(*R8 ------------------------*)
		(*Input Data*)
		R8.FB_In.Robot_Type:=KUKA_KRC4_SAFEOP;
		R8.FB_In.Install_Zero_Orientation:= 0; 	(*Set this value between 0 and 359 to set the zero position of the robot physical install with reference to 12 o'clock symbol on UI screens*)
		R8.FB_In.Under_Construction:= GTAC_CONFIG.Under_Construction;
		R8.FB_In.In_SIM_Mode:= GTAC_CONFIG.In_SIM_Mode;
		R8.FB_In.SIM_StartWorkAround:= FALSE;  (*Main.SIM_WorkAround_StartRobots*)
		R8.FB_In.CoE_Read_Trigger:= (GTAC_CONFIG.Option_Robot_Count>=8) AND Pulse_CoERead;
		R8.FB_In.Ecat_Master_AmsNetID:= MAIN.ECAT_Master.AmsID;
		R8.FB_In.Prev_EcatNode_Present:= NOT R7.EK1100_NotPresent; (*Ensure Previous Node Exists to determine Ecat Cable Break of this Devices Input Cable*)
		R8.FB_In.Safety_RST:=SAFETY_RESET;
		R8.FB_In.Enable_Motion:= All_Estops_OK OR GTAC_CONFIG.Under_Construction;
		R8.FB_In.Alarm_RST:=In_From_ICxx.ControlPower1;
		R8.FB_In.Select_Play:=FALSE;
		R8.FB_In.Select_Teach:=FALSE;
		R8.FB_In.Select_Remote:=FALSE;
		R8.FB_In.Start_Scan:=In_From_ICxx.StartRobots;
		R8.FB_In.Stop_Scan:=In_From_ICxx.StopRobots;
		R8.FB_In.Stop_Scan2:=FALSE;
		R8.FB_In.In_DryCycle:= GTAC_CONFIG.Dry_Cycle_Enabled;
		R8.FB_In.Low_Speed:= GTAC_CONFIG.Low_Speed_Enabled;
		R8.FB_In.Speed_Request:= In_From_ICxx.Global_Robot_Speed;
		R8.FB_In.Force_MasterTest_Req:= Cell_Services_Prog.Human_Reqs_MasterTest OR Cell_Services_Prog.A_Robot_Reqs_MasterTest;
		R8.FB_In.Force_BrakeTest_Req:= Cell_Services_Prog.Human_Reqs_BrakeTest OR Cell_Services_Prog.A_Robot_Reqs_BrakeTest;
		R8.FB_In.Major_Faults:= Faults.System_Major_Fault;
		R8.FB_In.Teach_Interlock:=R8_Data.Teach_Interlock;
		R8.FB_In.Weld_Inhibit:=In_From_ICxx.Rxx_Weld_Inhibit;
		R8.FB_In.Option_Disable_WaterFLT:= FALSE AND GTAC_CONFIG.Under_Construction OR (MAIN.R8.Task_ID_Ack=Tip_Change_EXT); (*Used to disable water fault if no water is present. use with caution*)
		R8.FB_In.OK_ToEnter_EquipInterf1:=R8_Data.OK_ToEnter_EquipInterf1;
		R8.FB_In.OK_ToEnter_EquipInterf2:=R8_Data.OK_ToEnter_EquipInterf2;
		R8.FB_In.OK_ToEnter_EquipInterf3:=R8_Data.OK_ToEnter_EquipInterf3;
		R8.FB_In.OK_ToEnter_EquipInterf4:=R8_Data.OK_ToEnter_EquipInterf4;
		R8.FB_In.OK_ToEnter_EquipInterf5:=R8_Data.OK_ToEnter_EquipInterf5;
		R8.FB_In.OK_ToEnter_EquipInterf6:=R8_Data.OK_ToEnter_EquipInterf6;
		R8.FB_In.OK_ToEnter_EquipInterf7:=R8_Data.OK_ToEnter_EquipInterf7;
		R8.FB_In.OK_ToEnter_EquipInterf8:=R8_Data.OK_ToEnter_EquipInterf8;
		R8.FB_In.OK_ToEnter_EquipInterf9:=R8_Data.OK_ToEnter_EquipInterf9;
		R8.FB_In.OK_ToEnter_HumanInterf1:=R8_Data.OK_ToEnter_HumanInterf1;
		R8.FB_In.OK_ToEnter_HumanInterf2:=R8_Data.OK_ToEnter_HumanInterf2;
		R8.FB_In.OK_ToEnter_HumanInterf3:=R8_Data.OK_ToEnter_HumanInterf3;
		R8.FB_In.OK_ToEnter_HumanInterf4:=R8_Data.OK_ToEnter_HumanInterf4;
		R8.FB_In.OK_ToEnter_HumanInterf5:=R8_Data.OK_ToEnter_HumanInterf5;
		R8.FB_In.OK_ToEnter_HumanInterf6:=R8_Data.OK_ToEnter_HumanInterf6;
		R8.FB_In.OK_ToEnter_HumanInterf7:=R8_Data.OK_ToEnter_HumanInterf7;
		R8.FB_In.OK_ToEnter_HumanInterf8:=R8_Data.OK_ToEnter_HumanInterf8;
		R8.FB_In.OK_ToEnter_RobotInterfs:= R8_Data.OK_ToEnter_RobotInterfs;
		R8.FB_In.Fix_ID:=R8_Data.Fix_ID[R8.Location_Index];
		R8.FB_In.Model_ID:=R8_Data.Model_ID[R8.Location_Index];
		R8.FB_In.Task_ID:=R8_Data.Task_ID[R8.Location_Index];
		R8.FB_In.Proceed_From_Pounce:=R8_Data.Proceed_From_Pounce[R8.Location_Index];
		R8.FB_In.Complete_Ack:=R8_Data.Complete_Ack[R8.Location_Index];
		R8.FB_In.PeripheralReq_Ack:=R8_Data.PeripheralReq_Ack[R8.Location_Index];
		R8.FB_In.AuxReq_Ack:=R8_Data.AuxReq_Ack[R8.Location_Index];
		R8.FB_In.User_Inputs.0:= FALSE;
		R8.FB_In.User_Inputs.1:= FALSE;
		R8.FB_In.User_Inputs.2:= FALSE;
		R8.FB_In.User_Inputs.3:= FALSE;
		R8.FB_In.User_Inputs.4:= FALSE;
		R8.FB_In.User_Inputs.5:= FALSE;
		R8.FB_In.User_Inputs.6:= FALSE;
		R8.FB_In.User_Inputs.7:= FALSE;
			(*Configure Options Amounts*)
			R8.FB_In.Options.WeldCont_Amount:= 0; 					(*Select amount of Spot Type Weld Controllers here (0 min, 4 max)*)
			R8.FB_In.Options.WaterStand_Amount:= 0;				(*Select amount of Water Stands here (0 min, 2 max)*)
			R8.FB_In.Options.MIGCont_Amount:= 1;					(*Select amount of MIG Type Weld Controllers here (0 min, 1 max)*)
			R8.FB_In.Options.Reamer_Amount:= 1;					(*Select amount of Tip Reamers here (0 min, 1 max)*)
			R8.FB_In.Options.EOAT_Amount:= 0;						(*Assign EOAT number to robot (0 min, 10 max)*)
			(*Configure Options Parameters*)
			
			R8.Reamer[1](
				(*FB Inputs*)
					Enable_Motion:= All_Estops_OK,
					Fronius_Ream:= TRUE,
                    Binzel_Ream:= FALSE,  (*optional*)
					
					Ream_REQ:= R8.Peripheral_Req.1 AND ((R8.Task_ID_Ack=Tip_Dress)OR (R8.In_T1 AND R8.Peripheral_Req.5)),
					Ream_Time:= T#2S,
					Ream_Clamp_Open:= R8.Reamer[1].N01.I.1,
					Spray_REQ:= R8.Peripheral_Req.2 AND ((R8.Task_ID_Ack=Tip_Dress)OR (R8.In_T1 AND R8.Peripheral_Req.5)),
					Spray_Time:= T#2S,
					F_WireCutter_REQ:= R8.Peripheral_Req.4 AND ((R8.Task_ID_Ack=Tip_Dress)OR (R8.In_T1 AND R8.Peripheral_Req.5)),
					F_WireCutter_Time:= T#1S,
					
				(*FB Outputs*)
					Reaming_Complete=> ,(*mapped in cell services*)
					(*The following are for Binzel type reamers only*)
					LifterUp_ACK=> , (*mapped in cell services*)
					Clamp_ACK=>,(*mapped in cell services*)
					Injector_ACK=> ,(*mapped in cell services*)
					WireCutter_ACK=> (*mapped in cell services*)
					);
			(*R8.Reamer[1](
				(*FB Inputs*)
					Enable_Motion:= All_Estops_OK,
					Fronius_Ream:= TRUE,
                    Binzel_Ream:= FALSE,  (*optional*)
					Ream_REQ:= R8.Peripheral_Req.5 AND (R8.Task_ID_Ack=Tip_Dress),

				(*FB Outputs*)
					Reaming_Complete=> ,(*mapped in cell services*)
					);*)
		(*Call Actual Object*)
		R8();
		(*Output Data*)
		Out_To_ICxx.Robot[8].Robot_Type:= R8.FB_In.Robot_Type;
		Out_To_ICxx.Robot[8].Status:= R8.Status;
		Out_To_ICxx.Robot[8].Axis_Data[1]:= R8.S_Axis_Pos_Raw;
		Out_To_ICxx.Robot[8].In_Image:= R8.Input_Image;
		Out_To_ICxx.Robot[8].Out_Image:= R8.Output_Image;
		Out_To_ICxx.Robot[8].Discrete_ImageFSOE:= R8.Discrete_Image_FSoE;
		Out_To_ICxx.Robot[8].Options:= R8.FB_In.Options;
			Out_To_ICxx.Robot[8].WS_Discrete_Image[1]:= R8.WS[1].Discrete_Image;
			Out_To_ICxx.Robot[8].WS_Discrete_Image[2]:= R8.WS[2].Discrete_Image;
 			Out_To_ICxx.Robot[8].ATI_Discrete_Image:= R8.ATI[1].Discrete_Image;
			Out_To_ICxx.Robot[8].Reamer_Discrete_Image:= R8.Reamer[1].Discrete_Image;
			Out_To_ICxx.Robot[8].Fronius_Status:= R8.Fronius_Status;
		Out_To_ICxx.Robot[8].Ped_IO_ToShow[1]:= 0;			(*Set to Ped value if this robots ecat string contains the Ped's IO*)
		Out_To_ICxx.Robot[8].Ped_IO_ToShow[2]:= 0;			(*Set to Ped value if this robots ecat string contains the Ped's IO*)
		Out_To_ICxx.Robot[8].ECAT_Cable_Breaks:= R8.ECatSlave_Cable_Breaks;
		Out_To_ICxx.Robot[8].CT:= R8.CT;



(*R9 ------------------------*)
		(*Input Data*)
		R9.FB_In.Robot_Type:=KUKA_KRC4_SAFEOP;
		R9.FB_In.Install_Zero_Orientation:= 0; 	(*Set this value between 0 and 359 to set the zero position of the robot physical install with reference to 12 o'clock symbol on UI screens*)
		R9.FB_In.Under_Construction:= GTAC_CONFIG.Under_Construction;
		R9.FB_In.In_SIM_Mode:= GTAC_CONFIG.In_SIM_Mode;
		R9.FB_In.SIM_StartWorkAround:= FALSE;  (*Main.SIM_WorkAround_StartRobots*)
		R9.FB_In.CoE_Read_Trigger:= (GTAC_CONFIG.Option_Robot_Count>=9) AND Pulse_CoERead;
		R9.FB_In.Ecat_Master_AmsNetID:= MAIN.ECAT_Master.AmsID;
		R9.FB_In.Prev_EcatNode_Present:= NOT R8.EK1100_NotPresent; (*Ensure Previous Node Exists to determine Ecat Cable Break of this Devices Input Cable*)
		R9.FB_In.Safety_RST:=SAFETY_RESET;
		R9.FB_In.Enable_Motion:= All_Estops_OK OR GTAC_CONFIG.Under_Construction;
		R9.FB_In.Alarm_RST:=In_From_ICxx.ControlPower1;
		R9.FB_In.Select_Play:=FALSE;
		R9.FB_In.Select_Teach:=FALSE;
		R9.FB_In.Select_Remote:=FALSE;
		R9.FB_In.Start_Scan:=In_From_ICxx.StartRobots;
		R9.FB_In.Stop_Scan:=In_From_ICxx.StopRobots;
		R9.FB_In.Stop_Scan2:=FALSE;
		R9.FB_In.In_DryCycle:= GTAC_CONFIG.Dry_Cycle_Enabled;
		R9.FB_In.Low_Speed:= GTAC_CONFIG.Low_Speed_Enabled;
		R9.FB_In.Speed_Request:= In_From_ICxx.Global_Robot_Speed;
		R9.FB_In.Force_MasterTest_Req:= Cell_Services_Prog.Human_Reqs_MasterTest OR Cell_Services_Prog.A_Robot_Reqs_MasterTest;
		R9.FB_In.Force_BrakeTest_Req:= Cell_Services_Prog.Human_Reqs_BrakeTest OR Cell_Services_Prog.A_Robot_Reqs_BrakeTest;
		R9.FB_In.Major_Faults:= Faults.System_Major_Fault;
		R9.FB_In.Teach_Interlock:=R9_Data.Teach_Interlock;
		R9.FB_In.Weld_Inhibit:=In_From_ICxx.Rxx_Weld_Inhibit;
		R9.FB_In.Option_Disable_WaterFLT:= FALSE AND GTAC_CONFIG.Under_Construction OR (MAIN.R9.Task_ID_Ack=Tip_Change_EXT); (*Used to disable water fault if no water is present. use with caution*)
		R9.FB_In.OK_ToEnter_EquipInterf1:=R9_Data.OK_ToEnter_EquipInterf1;
		R9.FB_In.OK_ToEnter_EquipInterf2:=R9_Data.OK_ToEnter_EquipInterf2;
		R9.FB_In.OK_ToEnter_EquipInterf3:=R9_Data.OK_ToEnter_EquipInterf3;
		R9.FB_In.OK_ToEnter_EquipInterf4:=R9_Data.OK_ToEnter_EquipInterf4;
		R9.FB_In.OK_ToEnter_EquipInterf5:=R9_Data.OK_ToEnter_EquipInterf5;
		R9.FB_In.OK_ToEnter_EquipInterf6:=R9_Data.OK_ToEnter_EquipInterf6;
		R9.FB_In.OK_ToEnter_EquipInterf7:=R9_Data.OK_ToEnter_EquipInterf7;
		R9.FB_In.OK_ToEnter_EquipInterf8:=R9_Data.OK_ToEnter_EquipInterf8;
		R9.FB_In.OK_ToEnter_EquipInterf9:=R9_Data.OK_ToEnter_EquipInterf9;
		R9.FB_In.OK_ToEnter_HumanInterf1:=R9_Data.OK_ToEnter_HumanInterf1;
		R9.FB_In.OK_ToEnter_HumanInterf2:=R9_Data.OK_ToEnter_HumanInterf2;
		R9.FB_In.OK_ToEnter_HumanInterf3:=R9_Data.OK_ToEnter_HumanInterf3;
		R9.FB_In.OK_ToEnter_HumanInterf4:=R9_Data.OK_ToEnter_HumanInterf4;
		R9.FB_In.OK_ToEnter_HumanInterf5:=R9_Data.OK_ToEnter_HumanInterf5;
		R9.FB_In.OK_ToEnter_HumanInterf6:=R9_Data.OK_ToEnter_HumanInterf6;
		R9.FB_In.OK_ToEnter_HumanInterf7:=R9_Data.OK_ToEnter_HumanInterf7;
		R9.FB_In.OK_ToEnter_HumanInterf8:=R9_Data.OK_ToEnter_HumanInterf8;
		R9.FB_In.OK_ToEnter_RobotInterfs:= R9_Data.OK_ToEnter_RobotInterfs;
		R9.FB_In.Fix_ID:=R9_Data.Fix_ID[R9.Location_Index];
		R9.FB_In.Model_ID:=R9_Data.Model_ID[R9.Location_Index];
		R9.FB_In.Task_ID:=R9_Data.Task_ID[R9.Location_Index];
		R9.FB_In.Proceed_From_Pounce:=R9_Data.Proceed_From_Pounce[R9.Location_Index];
		R9.FB_In.Complete_Ack:=R9_Data.Complete_Ack[R9.Location_Index];
		R9.FB_In.PeripheralReq_Ack:=R9_Data.PeripheralReq_Ack[R9.Location_Index];
		R9.FB_In.AuxReq_Ack:=R9_Data.AuxReq_Ack[R9.Location_Index];
		R9.FB_In.User_Inputs.0:= FALSE;
		R9.FB_In.User_Inputs.1:= FALSE;
		R9.FB_In.User_Inputs.2:= FALSE;
		R9.FB_In.User_Inputs.3:= FALSE;
		R9.FB_In.User_Inputs.4:= FALSE;
		R9.FB_In.User_Inputs.5:= FALSE;
		R9.FB_In.User_Inputs.6:= FALSE;
		R9.FB_In.User_Inputs.7:= FALSE;
			(*Configure Options Amounts*)
			R9.FB_In.Options.WeldCont_Amount:= 0; 					(*Select amount of Spot Type Weld Controllers here (0 min, 4 max)*)
			R9.FB_In.Options.WaterStand_Amount:= 0;				(*Select amount of Water Stands here (0 min, 2 max)*)
			R9.FB_In.Options.MIGCont_Amount:= 1;					(*Select amount of MIG Type Weld Controllers here (0 min, 1 max)*)
			R9.FB_In.Options.Reamer_Amount:= 1;					(*Select amount of Tip Reamers here (0 min, 1 max)*)
			R9.FB_In.Options.EOAT_Amount:= 0;						(*Assign EOAT number to robot (0 min, 10 max)*)
			(*Configure Options Parameters*)
			
			R9.Reamer[1](
				(*FB Inputs*)
					Enable_Motion:= All_Estops_OK,
					Fronius_Ream:= TRUE,
                    Binzel_Ream:= FALSE,  (*optional*)
					
					Ream_REQ:= R9.Peripheral_Req.1 AND ((R9.Task_ID_Ack=Tip_Dress)OR (R9.In_T1 AND R9.Peripheral_Req.5)),
					Ream_Time:= T#2S,
					Ream_Clamp_Open:= R9.Reamer[1].N01.I.1,
					Spray_REQ:= R9.Peripheral_Req.2 AND ((R9.Task_ID_Ack=Tip_Dress)OR (R9.In_T1 AND R9.Peripheral_Req.5)),
					Spray_Time:= T#2S,
					F_WireCutter_REQ:= R9.Peripheral_Req.4 AND ((R9.Task_ID_Ack=Tip_Dress)OR (R9.In_T1 AND R9.Peripheral_Req.5)),
					F_WireCutter_Time:= T#1S,
					
				(*FB Outputs*)
					Reaming_Complete=> ,(*mapped in cell services*)
					(*The following are for Binzel type reamers only*)
					LifterUp_ACK=> , (*mapped in cell services*)
					Clamp_ACK=>,(*mapped in cell services*)
					Injector_ACK=> ,(*mapped in cell services*)
					WireCutter_ACK=> (*mapped in cell services*)
					);
			(*R9.Reamer[1](
				(*FB Inputs*)
					Enable_Motion:= All_Estops_OK,
					Fronius_Ream:= TRUE,
                    Binzel_Ream:= FALSE,  (*optional*)
					Ream_REQ:= R9.Peripheral_Req.5 AND (R9.Task_ID_Ack=Tip_Dress),

				(*FB Outputs*)
					Reaming_Complete=> ,(*mapped in cell services*)
					);*)
		(*Call Actual Object*)
		R9();
		(*Output Data*)
		Out_To_ICxx.Robot[9].Robot_Type:= R9.FB_In.Robot_Type;
		Out_To_ICxx.Robot[9].Status:= R9.Status;
		Out_To_ICxx.Robot[9].Axis_Data[1]:= R9.S_Axis_Pos_Raw;
		Out_To_ICxx.Robot[9].In_Image:= R9.Input_Image;
		Out_To_ICxx.Robot[9].Out_Image:= R9.Output_Image;
		Out_To_ICxx.Robot[9].Discrete_ImageFSOE:= R9.Discrete_Image_FSoE;
		Out_To_ICxx.Robot[9].Options:= R9.FB_In.Options;
			Out_To_ICxx.Robot[9].WS_Discrete_Image[1]:= R9.WS[1].Discrete_Image;
			Out_To_ICxx.Robot[9].WS_Discrete_Image[2]:= R9.WS[2].Discrete_Image;
 			Out_To_ICxx.Robot[9].ATI_Discrete_Image:= R9.ATI[1].Discrete_Image;
			Out_To_ICxx.Robot[9].Reamer_Discrete_Image:= R9.Reamer[1].Discrete_Image;
			Out_To_ICxx.Robot[9].Fronius_Status:= R9.Fronius_Status;
		Out_To_ICxx.Robot[9].Ped_IO_ToShow[1]:= 0;			(*Set to Ped value if this robots ecat string contains the Ped's IO*)
		Out_To_ICxx.Robot[9].Ped_IO_ToShow[2]:= 0;			(*Set to Ped value if this robots ecat string contains the Ped's IO*)
		Out_To_ICxx.Robot[9].ECAT_Cable_Breaks:= R9.ECatSlave_Cable_Breaks;
		Out_To_ICxx.Robot[9].CT:= R9.CT;



(*R10 ------------------------*)
		(*Input Data*)
		R10.FB_In.Robot_Type:=KUKA_KRC4_SAFEOP;
		R10.FB_In.Install_Zero_Orientation:= 0; 	(*Set this value between 0 and 359 to set the zero position of the robot physical install with reference to 12 o'clock symbol on UI screens*)
		R10.FB_In.Under_Construction:= GTAC_CONFIG.Under_Construction;
		R10.FB_In.In_SIM_Mode:= GTAC_CONFIG.In_SIM_Mode;
		R10.FB_In.SIM_StartWorkAround:= FALSE;  (*Main.SIM_WorkAround_StartRobots*)
		R10.FB_In.CoE_Read_Trigger:= (GTAC_CONFIG.Option_Robot_Count>=10) AND Pulse_CoERead;
		R10.FB_In.Ecat_Master_AmsNetID:= MAIN.ECAT_Master.AmsID;
		R10.FB_In.Prev_EcatNode_Present:= NOT R9.EK1100_NotPresent; (*Ensure Previous Node Exists to determine Ecat Cable Break of this Devices Input Cable*)
		R10.FB_In.Safety_RST:=SAFETY_RESET;
		R10.FB_In.Enable_Motion:= All_Estops_OK OR GTAC_CONFIG.Under_Construction;
		R10.FB_In.Alarm_RST:=In_From_ICxx.ControlPower1;
		R10.FB_In.Select_Play:=FALSE;
		R10.FB_In.Select_Teach:=FALSE;
		R10.FB_In.Select_Remote:=FALSE;
		R10.FB_In.Start_Scan:=In_From_ICxx.StartRobots;
		R10.FB_In.Stop_Scan:=In_From_ICxx.StopRobots;
		R10.FB_In.Stop_Scan2:=FALSE;
		R10.FB_In.In_DryCycle:= GTAC_CONFIG.Dry_Cycle_Enabled;
		R10.FB_In.Low_Speed:= GTAC_CONFIG.Low_Speed_Enabled;
		R10.FB_In.Speed_Request:= In_From_ICxx.Global_Robot_Speed;
		R10.FB_In.Force_MasterTest_Req:= Cell_Services_Prog.Human_Reqs_MasterTest OR Cell_Services_Prog.A_Robot_Reqs_MasterTest;
		R10.FB_In.Force_BrakeTest_Req:= Cell_Services_Prog.Human_Reqs_BrakeTest OR Cell_Services_Prog.A_Robot_Reqs_BrakeTest;
		R10.FB_In.Major_Faults:= Faults.System_Major_Fault;
		R10.FB_In.Teach_Interlock:=R10_Data.Teach_Interlock;
		R10.FB_In.Weld_Inhibit:=In_From_ICxx.Rxx_Weld_Inhibit;
		R10.FB_In.Option_Disable_WaterFLT:= FALSE AND GTAC_CONFIG.Under_Construction OR (MAIN.R10.Task_ID_Ack=Tip_Change_EXT); (*Used to disable water fault if no water is present. use with caution*)
		R10.FB_In.OK_ToEnter_EquipInterf1:=R10_Data.OK_ToEnter_EquipInterf1;
		R10.FB_In.OK_ToEnter_EquipInterf2:=R10_Data.OK_ToEnter_EquipInterf2;
		R10.FB_In.OK_ToEnter_EquipInterf3:=R10_Data.OK_ToEnter_EquipInterf3;
		R10.FB_In.OK_ToEnter_EquipInterf4:=R10_Data.OK_ToEnter_EquipInterf4;
		R10.FB_In.OK_ToEnter_EquipInterf5:=R10_Data.OK_ToEnter_EquipInterf5;
		R10.FB_In.OK_ToEnter_EquipInterf6:=R10_Data.OK_ToEnter_EquipInterf6;
		R10.FB_In.OK_ToEnter_EquipInterf7:=R10_Data.OK_ToEnter_EquipInterf7;
		R10.FB_In.OK_ToEnter_EquipInterf8:=R10_Data.OK_ToEnter_EquipInterf8;
		R10.FB_In.OK_ToEnter_EquipInterf9:=R10_Data.OK_ToEnter_EquipInterf9;
		R10.FB_In.OK_ToEnter_HumanInterf1:=R10_Data.OK_ToEnter_HumanInterf1;
		R10.FB_In.OK_ToEnter_HumanInterf2:=R10_Data.OK_ToEnter_HumanInterf2;
		R10.FB_In.OK_ToEnter_HumanInterf3:=R10_Data.OK_ToEnter_HumanInterf3;
		R10.FB_In.OK_ToEnter_HumanInterf4:=R10_Data.OK_ToEnter_HumanInterf4;
		R10.FB_In.OK_ToEnter_HumanInterf5:=R10_Data.OK_ToEnter_HumanInterf5;
		R10.FB_In.OK_ToEnter_HumanInterf6:=R10_Data.OK_ToEnter_HumanInterf6;
		R10.FB_In.OK_ToEnter_HumanInterf7:=R10_Data.OK_ToEnter_HumanInterf7;
		R10.FB_In.OK_ToEnter_HumanInterf8:=R10_Data.OK_ToEnter_HumanInterf8;
		R10.FB_In.OK_ToEnter_RobotInterfs:= R10_Data.OK_ToEnter_RobotInterfs;
		R10.FB_In.Fix_ID:=R10_Data.Fix_ID[R10.Location_Index];
		R10.FB_In.Model_ID:=R10_Data.Model_ID[R10.Location_Index];
		R10.FB_In.Task_ID:=R10_Data.Task_ID[R10.Location_Index];
		R10.FB_In.Proceed_From_Pounce:=R10_Data.Proceed_From_Pounce[R10.Location_Index];
		R10.FB_In.Complete_Ack:=R10_Data.Complete_Ack[R10.Location_Index];
		R10.FB_In.PeripheralReq_Ack:=R10_Data.PeripheralReq_Ack[R10.Location_Index];
		R10.FB_In.AuxReq_Ack:=R10_Data.AuxReq_Ack[R10.Location_Index];
		R10.FB_In.User_Inputs.0:= FALSE;
		R10.FB_In.User_Inputs.1:= FALSE;
		R10.FB_In.User_Inputs.2:= FALSE;
		R10.FB_In.User_Inputs.3:= FALSE;
		R10.FB_In.User_Inputs.4:= FALSE;
		R10.FB_In.User_Inputs.5:= FALSE;
		R10.FB_In.User_Inputs.6:= FALSE;
		R10.FB_In.User_Inputs.7:= FALSE;
			(*Configure Options Amounts*)
			R10.FB_In.Options.WeldCont_Amount:= 0; 					(*Select amount of Spot Type Weld Controllers here (0 min, 4 max)*)
			R10.FB_In.Options.WaterStand_Amount:= 0;				(*Select amount of Water Stands here (0 min, 2 max)*)
			R10.FB_In.Options.MIGCont_Amount:= 1;					(*Select amount of MIG Type Weld Controllers here (0 min, 1 max)*)
			R10.FB_In.Options.Reamer_Amount:= 1;					(*Select amount of Tip Reamers here (0 min, 1 max)*)
			R10.FB_In.Options.EOAT_Amount:= 0;					(*Assign EOAT number to robot (0 min, 10 max)*)
			(*Configure Options Parameters*)
			(*R10.Reamer[1](
				(*FB Inputs*)
					Enable_Motion:= All_Estops_OK,
					Fronius_Ream:= TRUE,
                    Binzel_Ream:= FALSE,  (*optional*)
					Ream_REQ:= R10.Peripheral_Req.5 AND (R10.Task_ID_Ack=Tip_Dress),

				(*FB Outputs*)
					Reaming_Complete=> ,(*mapped in cell services*)
					);*)
		(*Call Actual Object*)
		R10();
		(*Output Data*)
		Out_To_ICxx.Robot[10].Robot_Type:= R10.FB_In.Robot_Type;
		(*To create less work, since there is no welding, changeing this number to 307 so we dont have to mess with the kuka FB, just screens. "us_Rxx_Status" - added 307 "inspecting"*)
		IF (R10.Status = 305) THEN
		Out_To_ICxx.Robot[10].Status:= 307; 
		ELSE
		Out_To_ICxx.Robot[10].Status:= R10.Status;
		END_IF
		Out_To_ICxx.Robot[10].Axis_Data[1]:= R10.S_Axis_Pos_Raw;
		Out_To_ICxx.Robot[10].In_Image:= R10.Input_Image;
		Out_To_ICxx.Robot[10].Out_Image:= R10.Output_Image;
		Out_To_ICxx.Robot[10].Discrete_ImageFSOE:= R10.Discrete_Image_FSoE;
		Out_To_ICxx.Robot[10].Options:= R10.FB_In.Options;
			Out_To_ICxx.Robot[10].WS_Discrete_Image[1]:= R10.WS[1].Discrete_Image;
			Out_To_ICxx.Robot[10].WS_Discrete_Image[2]:= R10.WS[2].Discrete_Image;
 			Out_To_ICxx.Robot[10].ATI_Discrete_Image:= R10.ATI[1].Discrete_Image;
			Out_To_ICxx.Robot[10].Reamer_Discrete_Image:= R10.Reamer[1].Discrete_Image;
			Out_To_ICxx.Robot[10].Fronius_Status:= R10.Fronius_Status;
		Out_To_ICxx.Robot[10].Ped_IO_ToShow[1]:= 0;			(*Set to Ped value if this robots ecat string contains the Ped's IO*)
		Out_To_ICxx.Robot[10].Ped_IO_ToShow[2]:= 0;			(*Set to Ped value if this robots ecat string contains the Ped's IO*)
		Out_To_ICxx.Robot[10].ECAT_Cable_Breaks:= R10.ECatSlave_Cable_Breaks;
		Out_To_ICxx.Robot[10].CT:= R10.CT;



(*R11 ------------------------*)
		(*Input Data*)
		R11.FB_In.Robot_Type:=KUKA_KRC4_SAFEOP;
		R11.FB_In.Install_Zero_Orientation:= 0; 	(*Set this value between 0 and 359 to set the zero position of the robot physical install with reference to 12 o'clock symbol on UI screens*)
		R11.FB_In.Under_Construction:= GTAC_CONFIG.Under_Construction;
		R11.FB_In.In_SIM_Mode:= GTAC_CONFIG.In_SIM_Mode;
		R11.FB_In.SIM_StartWorkAround:= FALSE;  (*Main.SIM_WorkAround_StartRobots*)
		R11.FB_In.CoE_Read_Trigger:= (GTAC_CONFIG.Option_Robot_Count>=11) AND Pulse_CoERead;
		R11.FB_In.Ecat_Master_AmsNetID:= MAIN.ECAT_Master.AmsID;
		R11.FB_In.Prev_EcatNode_Present:= NOT R10.EK1100_NotPresent; (*Ensure Previous Node Exists to determine Ecat Cable Break of this Devices Input Cable*)
		R11.FB_In.Safety_RST:=SAFETY_RESET;
		R11.FB_In.Enable_Motion:= All_Estops_OK OR GTAC_CONFIG.Under_Construction;
		R11.FB_In.Alarm_RST:=In_From_ICxx.ControlPower1;
		R11.FB_In.Select_Play:=FALSE;
		R11.FB_In.Select_Teach:=FALSE;
		R11.FB_In.Select_Remote:=FALSE;
		R11.FB_In.Start_Scan:=In_From_ICxx.StartRobots;
		R11.FB_In.Stop_Scan:=In_From_ICxx.StopRobots;
		R11.FB_In.Stop_Scan2:=FALSE;
		R11.FB_In.In_DryCycle:= GTAC_CONFIG.Dry_Cycle_Enabled;
		R11.FB_In.Low_Speed:= GTAC_CONFIG.Low_Speed_Enabled;
		R11.FB_In.Speed_Request:= In_From_ICxx.Global_Robot_Speed;
		R11.FB_In.Force_MasterTest_Req:= Cell_Services_Prog.Human_Reqs_MasterTest OR Cell_Services_Prog.A_Robot_Reqs_MasterTest;
		R11.FB_In.Force_BrakeTest_Req:= Cell_Services_Prog.Human_Reqs_BrakeTest OR Cell_Services_Prog.A_Robot_Reqs_BrakeTest;
		R11.FB_In.Major_Faults:= Faults.System_Major_Fault;
		R11.FB_In.Teach_Interlock:=R11_Data.Teach_Interlock;
		R11.FB_In.Weld_Inhibit:=In_From_ICxx.Rxx_Weld_Inhibit;
		R11.FB_In.Option_Disable_WaterFLT:= FALSE AND GTAC_CONFIG.Under_Construction OR (MAIN.R11.Task_ID_Ack=Tip_Change_EXT); (*Used to disable water fault if no water is present. use with caution*)
		R11.FB_In.OK_ToEnter_EquipInterf1:=R11_Data.OK_ToEnter_EquipInterf1;
		R11.FB_In.OK_ToEnter_EquipInterf2:=R11_Data.OK_ToEnter_EquipInterf2;
		R11.FB_In.OK_ToEnter_EquipInterf3:=R11_Data.OK_ToEnter_EquipInterf3;
		R11.FB_In.OK_ToEnter_EquipInterf4:=R11_Data.OK_ToEnter_EquipInterf4;
		R11.FB_In.OK_ToEnter_EquipInterf5:=R11_Data.OK_ToEnter_EquipInterf5;
		R11.FB_In.OK_ToEnter_EquipInterf6:=R11_Data.OK_ToEnter_EquipInterf6;
		R11.FB_In.OK_ToEnter_EquipInterf7:=R11_Data.OK_ToEnter_EquipInterf7;
		R11.FB_In.OK_ToEnter_EquipInterf8:=R11_Data.OK_ToEnter_EquipInterf8;
		R11.FB_In.OK_ToEnter_EquipInterf9:=R11_Data.OK_ToEnter_EquipInterf9;
		R11.FB_In.OK_ToEnter_HumanInterf1:=R11_Data.OK_ToEnter_HumanInterf1;
		R11.FB_In.OK_ToEnter_HumanInterf2:=R11_Data.OK_ToEnter_HumanInterf2;
		R11.FB_In.OK_ToEnter_HumanInterf3:=R11_Data.OK_ToEnter_HumanInterf3;
		R11.FB_In.OK_ToEnter_HumanInterf4:=R11_Data.OK_ToEnter_HumanInterf4;
		R11.FB_In.OK_ToEnter_HumanInterf5:=R11_Data.OK_ToEnter_HumanInterf5;
		R11.FB_In.OK_ToEnter_HumanInterf6:=R11_Data.OK_ToEnter_HumanInterf6;
		R11.FB_In.OK_ToEnter_HumanInterf7:=R11_Data.OK_ToEnter_HumanInterf7;
		R11.FB_In.OK_ToEnter_HumanInterf8:=R11_Data.OK_ToEnter_HumanInterf8;
		R11.FB_In.OK_ToEnter_RobotInterfs:= R11_Data.OK_ToEnter_RobotInterfs;
		R11.FB_In.Fix_ID:=R11_Data.Fix_ID[R11.Location_Index];
		R11.FB_In.Model_ID:=R11_Data.Model_ID[R11.Location_Index];
		R11.FB_In.Task_ID:=R11_Data.Task_ID[R11.Location_Index];
		R11.FB_In.Proceed_From_Pounce:=R11_Data.Proceed_From_Pounce[R11.Location_Index];
		R11.FB_In.Complete_Ack:=R11_Data.Complete_Ack[R11.Location_Index];
		R11.FB_In.PeripheralReq_Ack:=R11_Data.PeripheralReq_Ack[R11.Location_Index];
		R11.FB_In.AuxReq_Ack:=R11_Data.AuxReq_Ack[R11.Location_Index];
		R11.FB_In.User_Inputs.0:= FALSE;
		R11.FB_In.User_Inputs.1:= FALSE;
		R11.FB_In.User_Inputs.2:= FALSE;
		R11.FB_In.User_Inputs.3:= FALSE;
		R11.FB_In.User_Inputs.4:= FALSE;
		R11.FB_In.User_Inputs.5:= FALSE;
		R11.FB_In.User_Inputs.6:= FALSE;
		R11.FB_In.User_Inputs.7:= FALSE;
			(*Configure Options Amounts*)
			R11.FB_In.Options.WeldCont_Amount:= 0; 					(*Select amount of Spot Type Weld Controllers here (0 min, 4 max)*)
			R11.FB_In.Options.WaterStand_Amount:= 0;				(*Select amount of Water Stands here (0 min, 2 max)*)
			R11.FB_In.Options.MIGCont_Amount:= 1;					(*Select amount of MIG Type Weld Controllers here (0 min, 1 max)*)
			R11.FB_In.Options.Reamer_Amount:= 1;					(*Select amount of Tip Reamers here (0 min, 1 max)*)
			R11.FB_In.Options.EOAT_Amount:= 0;					(*Assign EOAT number to robot (0 min, 10 max)*)
			(*Configure Options Parameters*)
			(*R11.Reamer[1](
				(*FB Inputs*)
					Enable_Motion:= All_Estops_OK,
					Fronius_Ream:= TRUE,
                    Binzel_Ream:= FALSE,  (*optional*)
					Ream_REQ:= R11.Peripheral_Req.5 AND (R11.Task_ID_Ack=Tip_Dress),

				(*FB Outputs*)
					Reaming_Complete=> ,(*mapped in cell services*)
					);*)
		(*Call Actual Object*)
		R11();
		(*Output Data*)
		Out_To_ICxx.Robot[11].Robot_Type:= R11.FB_In.Robot_Type;
		(*To create less work, since there is no welding, changeing this number to 307 so we dont have to mess with the kuka FB, just screens. "us_Rxx_Status" - added 307 "inspecting"*)
		IF (R11.Status = 305) THEN
		Out_To_ICxx.Robot[11].Status:= 307; 
		ELSE
		Out_To_ICxx.Robot[11].Status:= R11.Status;
		END_IF
		Out_To_ICxx.Robot[11].Axis_Data[1]:= R11.S_Axis_Pos_Raw;
		Out_To_ICxx.Robot[11].In_Image:= R11.Input_Image;
		Out_To_ICxx.Robot[11].Out_Image:= R11.Output_Image;
		Out_To_ICxx.Robot[11].Discrete_ImageFSOE:= R11.Discrete_Image_FSoE;
		Out_To_ICxx.Robot[11].Options:= R11.FB_In.Options;
			Out_To_ICxx.Robot[11].WS_Discrete_Image[1]:= R11.WS[1].Discrete_Image;
			Out_To_ICxx.Robot[11].WS_Discrete_Image[2]:= R11.WS[2].Discrete_Image;
 			Out_To_ICxx.Robot[11].ATI_Discrete_Image:= R11.ATI[1].Discrete_Image;
			Out_To_ICxx.Robot[11].Reamer_Discrete_Image:= R11.Reamer[1].Discrete_Image;
			Out_To_ICxx.Robot[11].Fronius_Status:= R11.Fronius_Status;
		Out_To_ICxx.Robot[11].Ped_IO_ToShow[1]:= 0;			(*Set to Ped value if this robots ecat string contains the Ped's IO*)
		Out_To_ICxx.Robot[11].Ped_IO_ToShow[2]:= 0;			(*Set to Ped value if this robots ecat string contains the Ped's IO*)
		Out_To_ICxx.Robot[11].ECAT_Cable_Breaks:= R11.ECatSlave_Cable_Breaks;
		Out_To_ICxx.Robot[11].CT:= R11.CT;























(*end*)
END_ACTION

// ---- POUs/FBs/FB_GTAC_EtherCATMaster_20250723.TcPOU
(*FB for use as Instance of EtherCat Master

	Original Author(s): B.Lekx-Toniolo of Sodecia GTAC.; 
------------------------------------------------------------------------------------------
REVISION NOTES:
	Version 20160407
		- intial concept, b.lekx-toniolo
	Version 20160803
		- added SDxx (Servo Drive) component type for HW read, b.lekx-toniolo
	Version 20161116
		- Corrected bug to provide more room for overridables, b.lekx-toniolo
	Version 20170309
		- Increased largest readable slave count from 500 to 510, b.lekx-toniolo
	Version 20190925
		- Increased largest readable slave count from 510 to 800, b.lekx-toniolo
		- Added Maximum_Permissable_Slaves variable to be able to staticly set max from one location, b.lekx-toniolo
		- Add Config_SlaveCount_ExceedsMax_FLT variable as a fault flag for capturing maximum slave count exceeded, b.lekx-toniolo
	Version 20191127
		- Changed input of CoE_ReadConfFB_1.cbBufLen from static value to Sizeof value to provide compatibility with 
		  TC build 2305 forward (previous builds didn't regard the value of this input), b.lekx-toniolo
		- Moved Maximum_Permissable_Slaves to VAR CONSTANT area and also used as upper bounds while declaring of  CoE_ReadConfBuffer_1 array 
			(to further automate configurability of the code)
	Version 20220224
		- Changes during TcUI migration project, b.lekx-toniolo / c.drees
	Version 20250205
		- Re-wrote Auto Fixture code and integrated into old standard code (for Fixtures, EOATs and PEDs), b.lekx-toniolo 
		- See SSCC610 GH Issue #191 for more details, b.lekx-toniolo
	Version 20250723
		- Adeed in code to captue VFD type component, b.lekx-toniolo 

------------------------------------------------------------------------------------------
*)



FUNCTION_BLOCK FB_GTAC_EtherCATMaster_20250723
VAR_INPUT
	Enable_FB: BOOL;
	Blank_Config_Trigger: BOOL;
	Read_Config_Trigger: BOOL;
	Read_States_Trigger: BOOL;
	Machine_Running: BOOL;
	ComponentConfig_Overrides: ARRAY [0..100] OF STRING[5];								(*Storage Area for Configuration Overrides*)
END_VAR



VAR CONSTANT
	(*Set Some System limits*)
	(*USE CAUTION setting this value, if you're unsure what this value should and can be set to, do not touch, b.lekx-toniolo*)
	Maximum_Permissable_Slaves: UINT := 800;				(*Set's COE slave count read limit*)

END_VAR

VAR
(*Establish Data Area for EtherCAT Master Status Information*)
		HW_Status AT %I*: udt_ECATMaster_Status_20141211;
		AmsID_FB: FB_FormatString;	(*FB to assemble and output string from AMS Net ID Array*)
(*CoE Read*)
		CoE_ReadConfFB_1: FB_EcGetConfSlaves; 												(*FB to retrieve Configured Slave Data from ECAT Master*)
		CoE_ReadConfBuffer_1: ARRAY[0..Maximum_Permissable_Slaves] OF ST_EcSlaveConfigData;	(*Buffer (size configured by constant above), for receiving data*)
		CoE_ReadConfBuffer_LastRead: ARRAY[0..Maximum_Permissable_Slaves] OF ST_EcSlaveConfigData;	(*Buffer (size configured by constant above), for receiving data*)
		CoE_ReadConfErr_1: BOOL;															(*CoE Read Error Flag*)
		CoE_ReadConfErrID_1: UDINT;															(*CoE Read Error Identification*)
		CoE_NumberOfSlaves: UINT;															(*CoE Read Number of Slaves found in config*)
		ReadConf_DoneTRIG: R_TRIG;
		CaptureConf_TRIG: R_TRIG;
		
	
		CoE_ReadStatesFB_1: FB_EcGetAllSlaveStates; 												(*FB to retrieve Configured Slave Data from ECAT Master*)
		CoE_ReadStatesBuffer_1: ARRAY[0..Maximum_Permissable_Slaves] OF ST_EcSlaveState;	(*Buffer (size configured by constant above), for receiving data*)
		CoE_ReadStatesBuffer_LastRead: ARRAY[0..Maximum_Permissable_Slaves] OF ST_EcSlaveState;	(*Buffer (size configured by constant above), for receiving data*)
		CoE_ReadStatesErr_1: BOOL;															(*CoE Read Error Flag*)
		CoE_ReadStatesErrID_1: UDINT;															(*CoE Read Error Identification*)	
		ReadStates_DoneTRIG: R_TRIG;


		GTAC_ECAT_ComponentConfig: ARRAY [0..100] OF STRING[5];								(*Storage Area for Actual GTAC Component Based Config*)

		Build_ComponentConfig_Index: UINT;
		Blank_ComponentArray_Index: UINT;
		ComponentConfigArray_Index: UINT;
		Period_Position: INT;
		Component_Num_AsString: STRING(10);
		Component_Num_AsUINT: UINT;
		Config_SlaveCount_ExceedsMax_FLT: BOOL;											(*Flag if Hardware Config Slave count exceeds maximum for this FB*)
	
(*Areas and vars for building I/O Node Layouts*)	
		FixConfPointer :ARRAY[0..120] OF INT; 											(*Pointer for storing Fixture Data*)
		EOATConfPointer :ARRAY[0..30] OF INT; 											(*Pointer for storing Fixture Data*)
		PedConfPointer :ARRAY[0..30] OF INT; 											(*Pointer for storing Fixture Data*)

		FixNodeLayout :ARRAY[0..120] OF udt_ECATNodeData_20221507;					(*Data Area for Ped as Ped is an FB*)
		EOATNodeLayout :ARRAY[0..30] OF udt_ECATNodeData_20221507;					(*Data Area for Ped as Ped is an FB*)
		PedNodeLayout :ARRAY[0..30] OF udt_ECATNodeData_20221507;					(*Data Area for Ped as Ped is an FB*)


(*Node Model Setup*)
	InputNode: STRING:= 'EP1008';
	OutputNode: STRING:='EP2028';
	ValveBank: STRING:= 'EX260-';
	WSNode:STRING:= 'EP3172';
	NodeType: INT;
END_VAR

VAR_OUTPUT
		FB_OK: BOOL;
		AmsID: STRING;
		Discrete_Image: udt_ECATMaster_Image_20220224; 	(*Image Framework for EtherCAT Master Status*)
		(*Discrete Data for Fixtures *)
END_VAR

	(*Set FB_OK to True*)
	FB_OK:= TRUE;

(*$$$$$$$$$$$$$$$$$$$$$$$$$$$$$$$$$$$$$$$$$$$$$$$$Gather Status Of Hardware $$$$$$$$$$$$$$$$$$$$$$$$$$$$$$$$$$$$$$$$$$$$$$$$$$$$*)

(*$$$$$$$$$$$$$$$$$$$$$$$$$$$$$$$$$$$$$$$$$$$$$ Gather Safety Inputs $$$$$$$$$$$$$$$$$$$$$$$$$$$$$$$$$$$$$$$$$$$$$$$$$$$$$$$$$*)


(*$$$$$$$$$$$$$$$$$$$$$$$$$$$$$$$$$$$$$$$$$$$$$ Gather Standard Inputs $$$$$$$$$$$$$$$$$$$$$$$$$$$$$$$$$$$$$$$$$$$$$$$$$$$$$$$$$*)

(*$$$$$$$$$$$$$$$$$$$$$$$$$$$$$$$$$$$$$$$$$$$$$ Internal Code $$$$$$$$$$$$$$$$$$$$$$$$$$$$$$$$$$$$$$$$$$$$$$$$$$$$$$$$$*)

	(*Convert raw AMS Net ID data to a string*)
	(*Inputs*)
	AmsID_FB.sFormat:= '%u.%u.%u.%u.%u.%u';
	AmsID_FB.arg1:= F_USINT(HW_Status.Infodata.AmsNetId[0]);
	AmsID_FB.arg2:= F_USINT(HW_Status.Infodata.AmsNetId[1]);
	AmsID_FB.arg3:= F_USINT(HW_Status.Infodata.AmsNetId[2]);
	AmsID_FB.arg4:= F_USINT(HW_Status.Infodata.AmsNetId[3]);
	AmsID_FB.arg5:= F_USINT(HW_Status.Infodata.AmsNetId[4]);
	AmsID_FB.arg6:= F_USINT(HW_Status.Infodata.AmsNetId[5]);
	(*Actual Call to FB*)
	AmsID_FB();
	(*Outputs*)
	AmsID:= AmsID_FB.sOut;			(*Expose Output String*)


	(*------------ CoE Read (Slave Configs) ------------*)

	(*Read Through Slave Configuration data stored in EtherCAT Master*)

	(*FB Inputs*)
	CoE_ReadConfFB_1.bExecute:= (NOT Machine_Running AND Read_Config_Trigger) OR COE_ReadConfFB_1.bBusy;		(*Execute Upon Trigger*)
	CoE_ReadConfFB_1.sNetId:= AmsID;													(*AMS Address to EtherCAT Master*)
	CoE_ReadConfFB_1.cbBufLen:= SIZEOF(CoE_ReadConfBuffer_1);						(*Limit on Receive Length (bytes)*)
	CoE_ReadConfFB_1.pArrEcConfSlaveInfo:= ADR(CoE_ReadConfBuffer_1);					(*Pointer to Receive Buffer*)
	CoE_ReadConfFB_1.tTimeout:= T#3s;												(*TImeout for Read (used static value instead of standard ADS CONST to minimize external dependancies)*)

	(*Execute FB*)
	CoE_ReadConfFB_1();
	
	(*FB Outputs*)
	CoE_ReadConfErr_1:= CoE_ReadConfFB_1.bError;										(*Error Flag of Read*)
	CoE_ReadConfErrID_1:= CoE_ReadConfFB_1.nErrorId;									(*Error ID of Read (See ADS Return Codes)*)
	CoE_NumberOFSlaves:= CoE_ReadConfFB_1.nSlaves;									(*General Count of Slaves In HW Configuration*)

	(*Caputre Last Configuration Read*)
	ReadConf_DoneTRIG.CLK:= NOT CoE_ReadConfFB_1.bExecute;
	ReadConf_DoneTRIG();
	IF ReadConf_DoneTRIG.Q
		THEN
		CoE_ReadConfBuffer_LastRead:= CoE_ReadConfBuffer_1;
	END_IF
	
	(*------------ CoE Read (Slave States)------------*)

	(*Read Through Slave State data stored in EtherCAT Master*)

	(*FB Inputs*)
	CoE_ReadStatesFB_1.bExecute:= Read_States_Trigger OR CoE_ReadStatesFB_1.bBusy;		(*Execute Upon Trigger*)
	CoE_ReadStatesFB_1.sNetId:= AmsID;													(*AMS Address to EtherCAT Master*)
	CoE_ReadStatesFB_1.cbBufLen:= SIZEOF(CoE_ReadStatesBuffer_1);						(*Limit on Receive Length (bytes)*)
	CoE_ReadStatesFB_1.pStateBuf:= ADR(CoE_ReadStatesBuffer_1);						(*Pointer to Receive Buffer*)
	CoE_ReadStatesFB_1.tTimeout:= T#3S;												(*TImeout for Read (used static value instead of standard ADS CONST to minimize external dependancies)*)

	(*Execute FB*)
	CoE_ReadStatesFB_1();

	(*FB Outputs*)
	CoE_ReadStatesErr_1:= CoE_ReadStatesFB_1.bError;										(*Error Flag of Read*)
	CoE_ReadStatesErrID_1:= CoE_ReadStatesFB_1.nErrId;									(*Error ID of Read (See ADS Return Codes)*)

	(*Caputre Last States Read*)
	ReadStates_DoneTRIG.CLK:= NOT CoE_ReadConfFB_1.bExecute;
	ReadStates_DoneTRIG();
	IF ReadStates_DoneTRIG.Q
		THEN
		CoE_ReadStatesBuffer_LastRead:= CoE_ReadStatesBuffer_1;
	END_IF

(*-------------------------------------------------------------------------- Blank Config -----------------------------------------------------*)
	IF Blank_Config_Trigger OR Config_SlaveCount_ExceedsMax_FLT
		THEN
		FOR Blank_ComponentArray_Index:= 1 TO 100 DO
			GTAC_ECAT_ComponentConfig[Blank_ComponentArray_Index]:='';
		END_FOR;
	END_IF;

(*----------------------------------- Loop through Last CoE Read Slaves Configured and find GTAC Components -----------------------------*)
(*------------------------------------------------ Also parse out Associated State Values at same time ----------------------------------*)
	CaptureConf_TRIG.CLK:= NOT Blank_Config_Trigger AND NOT Read_States_Trigger;
	CaptureConf_TRIG();
	
	IF CaptureConf_TRIG.Q AND (CoE_NumberOfSlaves<=Maximum_Permissable_Slaves)
		THEN
		ComponentConfigArray_Index:= 1; 		(*Reset Config Array Index*)
		Period_Position:=0;
		Component_Num_AsString:= '';
		Component_Num_AsUINT:= 0;
		Config_SlaveCount_ExceedsMax_FLT:= FALSE;	(*Slave Count in Hardware Configuration is under Maximum Allowable by this FB so reset flag*)

		(*----------------- Loop through each Slave and evaluate what it is ----------------------------*)
		FOR Build_ComponentConfig_Index:= 0 TO CoE_NumberOfSlaves+1 DO
			
			(*------------------ First Check for Manual Configuration Overrdes ------------------------*)
			IF ComponentConfig_Overrides[ComponentConfigArray_Index]<>''
				THEN
				GTAC_ECAT_ComponentConfig[ComponentConfigArray_Index]:= FUN_GTAC_ReturnSetLengthSTR(
																			ComponentConfig_Overrides[ComponentConfigArray_Index], 5);
				ComponentConfigArray_Index:= ComponentConfigArray_Index+1;			(*Index to next element in Config Array*)

			(*---------- Caputre EK1100 Based Componenets ------------------------*)
			ELSIF FUN_GTAC_ReturnSetLengthSTR(CoE_ReadConfBuffer_LastRead[Build_ComponentConfig_Index].sType,6) = 'EK1100'
				THEN
				Period_Position:= FIND(CoE_ReadConfBuffer_LastRead[Build_ComponentConfig_Index].sName, '.');
				GTAC_ECAT_ComponentConfig[ComponentConfigArray_Index]:= FUN_GTAC_ReturnSetLengthSTR(
																				CoE_ReadConfBuffer_LastRead[Build_ComponentConfig_Index].sName, (Period_Position-1));
				ComponentConfigArray_Index:= ComponentConfigArray_Index+1;			(*Index to next element in Config Array*)

			(*----------------- Caputre MDxx Componenets ------------------------*)
			ELSIF FUN_GTAC_ReturnSetLengthSTR(CoE_ReadConfBuffer_LastRead[Build_ComponentConfig_Index].sType,6) = 'EP1918'
				THEN
				GTAC_ECAT_ComponentConfig[ComponentConfigArray_Index]:= FUN_GTAC_ReturnSetLengthSTR(
																			CoE_ReadConfBuffer_LastRead[Build_ComponentConfig_Index].sName, 4);
				ComponentConfigArray_Index:= ComponentConfigArray_Index+1;			(*Index to next element in Config Array*)

			(*----------------- Caputre ESWxx Componenets ------------------------*)
			ELSIF FUN_GTAC_ReturnSetLengthSTR(CoE_ReadConfBuffer_LastRead[Build_ComponentConfig_Index].sType,6) = 'EP1908'
				THEN
				GTAC_ECAT_ComponentConfig[ComponentConfigArray_Index]:= FUN_GTAC_ReturnSetLengthSTR(
																			CoE_ReadConfBuffer_LastRead[Build_ComponentConfig_Index].sName, 5);
				ComponentConfigArray_Index:= ComponentConfigArray_Index+1;			(*Index to next element in Config Array*)

			(*------------------ Caputre SSxx Componenets ------------------------*)
			ELSIF 	FUN_GTAC_ReturnSetLengthSTR(CoE_ReadConfBuffer_LastRead[Build_ComponentConfig_Index].sType,6) = 'EP9128'
				AND FUN_GTAC_ReturnSetLengthSTR(CoE_ReadConfBuffer_LastRead[Build_ComponentConfig_Index].sName,1) = 'S'

				THEN
				GTAC_ECAT_ComponentConfig[ComponentConfigArray_Index]:= FUN_GTAC_ReturnSetLengthSTR(
																			CoE_ReadConfBuffer_LastRead[Build_ComponentConfig_Index].sName, 4);
				ComponentConfigArray_Index:= ComponentConfigArray_Index+1;			(*Index to next element in Config Array*)
			(*---------- Caputre AX52xx Based Componenets ------------------------*)
			ELSIF FUN_GTAC_ReturnSetLengthSTR(CoE_ReadConfBuffer_LastRead[Build_ComponentConfig_Index].sType,4) = 'AX52'
				THEN
				Period_Position:= FIND(CoE_ReadConfBuffer_LastRead[Build_ComponentConfig_Index].sName, ' '); (*Actually a space position*)
				
				GTAC_ECAT_ComponentConfig[ComponentConfigArray_Index]:= FUN_GTAC_ReturnSetLengthSTR(
																				CoE_ReadConfBuffer_LastRead[Build_ComponentConfig_Index].sName, Period_Position -1);
				ComponentConfigArray_Index:= ComponentConfigArray_Index+1;			(*Index to next element in Config Array*)

			(*----------------- Caputre VFDxx Componenets ------------------------*)
			ELSIF FUN_GTAC_ReturnSetLengthSTR(CoE_ReadConfBuffer_LastRead[Build_ComponentConfig_Index].sType,6) = 'ATV320'
				THEN
				GTAC_ECAT_ComponentConfig[ComponentConfigArray_Index]:= FUN_GTAC_ReturnSetLengthSTR(
																			CoE_ReadConfBuffer_LastRead[Build_ComponentConfig_Index].sName, 5);
				ComponentConfigArray_Index:= ComponentConfigArray_Index+1;			(*Index to next element in Config Array*)

				
			(*---------- Caputre Fixture Based Components and Build Node Layout------------------------*)
			ELSIF FUN_GTAC_ReturnSetLengthSTR(CoE_ReadConfBuffer_LastRead[Build_ComponentConfig_Index].sName,3) = 'Fix'
				THEN
				Component_Num_AsString:= MID(CoE_ReadConfBuffer_LastRead[Build_ComponentConfig_Index].sName,3,4); (*Get Component Number*)
				Component_Num_AsUINT:= STRING_TO_UINT(Component_Num_AsString);
					FixNodeLayout[Component_Num_AsUINT].NodeType[FixConfPointer[Component_Num_AsUINT]]:= FUN_GTAC_ReturnSetLengthSTR(CoE_ReadConfBuffer_LastRead[Build_ComponentConfig_Index].sType,6);
					FixNodeLayout[Component_Num_AsUINT].NodeName[FixConfPointer[Component_Num_AsUINT]]:= CoE_ReadConfBuffer_LastRead[Build_ComponentConfig_Index].sName;
					FixNodeLayout[Component_Num_AsUINT].State[FixConfPointer[Component_Num_AsUINT]]:= INT_TO_UINT(FUN_GTAC_BYTEStoINT(CoE_ReadStatesBuffer_LastRead[Build_ComponentConfig_Index].deviceState,CoE_ReadStatesBuffer_LastRead[Build_ComponentConfig_Index].linkState));
				FixConfPointer[Component_Num_AsUINT]:= FixConfPointer[Component_Num_AsUINT]+1;
			(*---------- Caputre EOAT Based Components and Build Node Layout ------------------------*)
			ELSIF FUN_GTAC_ReturnSetLengthSTR(CoE_ReadConfBuffer_LastRead[Build_ComponentConfig_Index].sName,4) = 'EOAT'
				THEN
				Component_Num_AsString:= MID(CoE_ReadConfBuffer_LastRead[Build_ComponentConfig_Index].sName,2,5); (*Get Component Number*)
				Component_Num_AsUINT:= STRING_TO_UINT(Component_Num_AsString);
					EOATNodeLayout[Component_Num_AsUINT].NodeType[EOATConfPointer[Component_Num_AsUINT]]:= FUN_GTAC_ReturnSetLengthSTR(CoE_ReadConfBuffer_LastRead[Build_ComponentConfig_Index].sType,6);
					EOATNodeLayout[Component_Num_AsUINT].NodeName[EOATConfPointer[Component_Num_AsUINT]]:= CoE_ReadConfBuffer_LastRead[Build_ComponentConfig_Index].sName;
					EOATNodeLayout[Component_Num_AsUINT].State[EOATConfPointer[Component_Num_AsUINT]]:= INT_TO_UINT(FUN_GTAC_BYTEStoINT(CoE_ReadStatesBuffer_LastRead[Build_ComponentConfig_Index].deviceState,CoE_ReadStatesBuffer_LastRead[Build_ComponentConfig_Index].linkState));
				EOATConfPointer[Component_Num_AsUINT]:= EOATConfPointer[Component_Num_AsUINT]+1;
			(*---------- Caputre Ped Based Components and Build Node Layout ------------------------*)
			ELSIF FUN_GTAC_ReturnSetLengthSTR(CoE_ReadConfBuffer_LastRead[Build_ComponentConfig_Index].sName,3) = 'PED'
				THEN
				Component_Num_AsString:= MID(CoE_ReadConfBuffer_LastRead[Build_ComponentConfig_Index].sName,2,4); (*Get Component Number*)
				Component_Num_AsUINT:= STRING_TO_UINT(Component_Num_AsString);
					PedNodeLayout[Component_Num_AsUINT].NodeType[PedConfPointer[Component_Num_AsUINT]]:= FUN_GTAC_ReturnSetLengthSTR(CoE_ReadConfBuffer_LastRead[Build_ComponentConfig_Index].sType,6);
					PedNodeLayout[Component_Num_AsUINT].NodeName[PedConfPointer[Component_Num_AsUINT]]:= CoE_ReadConfBuffer_LastRead[Build_ComponentConfig_Index].sName;
					PedNodeLayout[Component_Num_AsUINT].State[PedConfPointer[Component_Num_AsUINT]]:= INT_TO_UINT(FUN_GTAC_BYTEStoINT(CoE_ReadStatesBuffer_LastRead[Build_ComponentConfig_Index].deviceState,CoE_ReadStatesBuffer_LastRead[Build_ComponentConfig_Index].linkState));
				PedConfPointer[Component_Num_AsUINT]:= PedConfPointer[Component_Num_AsUINT]+1;
			

			(*------------------ Default, blank data ----------------*)
			ELSE
				GTAC_ECAT_ComponentConfig[ComponentConfigArray_Index]:='';
			END_IF;

			(*Bounding protection*)
			IF ComponentConfigArray_Index>=100
				THEN
				ComponentConfigArray_Index:=100;
			END_IF;


		END_FOR; (*End Read Slave Config For loop*)
		
		(*Reset Node Layout Pointers at end of Slave evaluation to avoid continuous building of images*)
			MEMSET(ADR(FixConfPointer), 0, SIZEOF(FixConfPointer));
			MEMSET(ADR(EOATConfPointer), 0, SIZEOF(EOATConfPointer));
			MEMSET(ADR(PedConfPointer), 0, SIZEOF(PedConfPointer));


	ELSIF CoE_NumberOfSlaves>Maximum_Permissable_Slaves
		THEN
		Config_SlaveCount_ExceedsMax_FLT:= TRUE;	(*Slave Count in Hardware Configuration Exceeds Maximum Allowable by this FB, must consult b.lekx-toniolo if this happens*)
	END_IF;

	
	
(*????????????????????????????????????????????????????????????????????????????????????????????????????????????????*)

(*$$$$$$$$$$$$$$$$$$$$$$$$$$$$$$$$$$$$$$$$$$$$$$$$$$$ Faults $$$$$$$$$$$$$$$$$$$$$$$$$$$$$$$$$$$$$$$$$$$$$$$$$$$$$$$*)

(*$$$$$$$$$$$$$$$$$$$$$$$$$$$$$$$$$$$$$$$$$$$$$$ Transfer Standard Outputs $$$$$$$$$$$$$$$$$$$$$$$$$$$$$$$$$$$$$$$$$$$*)
	(*Transfer Image for display on UI*)
		Discrete_Image.HW:= HW_Status;
		Discrete_Image.AMS_ID:= AMSID;
		Discrete_Image.Config:=GTAC_ECAT_ComponentConfig;


(*$$$$$$$$$$$$$$$$$$$$$$$$$$$$$$$$$$$$$$$$$$$$$$ Transfer Safety Outputs $$$$$$$$$$$$$$$$$$$$$$$$$$$$$$$$$$$$$$$$$$$*)

END_FUNCTION_BLOCK

// ---- POUs/FUNs/FUN_GTAC_ReturnSetLengthSTR.TcPOU
(*Function to return a portion of source string (from a provided string) based on return length specified (starting at element 0 of source)
	author: Brent Lekx-Toniolo OF Sodecia GTAC
	date: April 2016
	version 1.0
		- initial concept


	Last Edit: 14-Oct-2021, BLT, added ability to return length of 22 (for a specific case)

*)

FUNCTION FUN_GTAC_ReturnSetLengthSTR : STRING
VAR_INPUT
	Source_String: STRING;
	Return_Length: UINT;

END_VAR
VAR
	String_Len1: STRING[1];
	String_Len2: STRING[2];
	String_Len3: STRING[3];
	String_Len4: STRING[4];
	String_Len5: STRING[5];
	String_Len6: STRING[6];
	String_Len7: STRING[7];
	String_Len8: STRING[8];
	String_Len9: STRING[9];
	String_Len10: STRING[10];
	String_Len21: STRING[21];
	String_Len22: STRING[22];

END_VAR

(*Return String Based on Length Requested*)

	CASE Return_Length OF
		1:
			String_Len1:= Source_String;
			FUN_GTAC_ReturnSetLengthSTR:= String_Len1;
	 	2:
			String_Len2:= Source_String;
			FUN_GTAC_ReturnSetLengthSTR:= String_Len2;
		3:
			String_Len3:= Source_String;
			FUN_GTAC_ReturnSetLengthSTR:= String_Len3;
		4:
			String_Len4:= Source_String;
			FUN_GTAC_ReturnSetLengthSTR:= String_Len4;
		5:
			String_Len5:= Source_String;
			FUN_GTAC_ReturnSetLengthSTR:= String_Len5;
		6:
			String_Len6:= Source_String;
			FUN_GTAC_ReturnSetLengthSTR:= String_Len6;
		7:
			String_Len7:= Source_String;
			FUN_GTAC_ReturnSetLengthSTR:= String_Len7;
		8:
			String_Len8:= Source_String;
			FUN_GTAC_ReturnSetLengthSTR:= String_Len8;
		9:
			String_Len9:= Source_String;
			FUN_GTAC_ReturnSetLengthSTR:= String_Len9;
		10:
			String_Len10:= Source_String;
			FUN_GTAC_ReturnSetLengthSTR:= String_Len10;	
		21:
			(*Sepecific case created for returning Machine serial parsed from TC3 Appname data*)
			String_Len21:= Source_String;
			FUN_GTAC_ReturnSetLengthSTR:= String_Len21;
		22:
			(*Sepecific case created for returning Machine serial parsed from TC3 Appname data, after serial number -> eng project number changes*)
			String_Len22:= Source_String;
			FUN_GTAC_ReturnSetLengthSTR:= String_Len22;


	 ELSE
		(*default case, blank return*)
			FUN_GTAC_ReturnSetLengthSTR:= '';

	END_CASE;

END_FUNCTION

// ---- POUs/FUNs/FUN_GTAC_BYTEStoINT.TcPOU
(*Copy Individual Bytes (input to the FUN) at bit level, into individual bits of the INT Return
	author: Brent Lekx-Toniolo OF Sodecia GTAC
	date: November 2012
	version 1.0
		- initial concept
	Last Edit: December 4th, 2012, BLT
*)

FUNCTION FUN_GTAC_BYTEStoINT : INT
VAR_INPUT
	Byte0: BYTE;
	Byte1: BYTE;
END_VAR
VAR
END_VAR

(*Copy Individual Bytes (input to the FUN) at bit level, into individual bits of the INT Return*)

(*Byte 0 to Lower 8 bits of Int*)
FUN_GTAC_BYTEStoINT.0:= Byte0.0;
FUN_GTAC_BYTEStoINT.1:= Byte0.1;
FUN_GTAC_BYTEStoINT.2:= Byte0.2;
FUN_GTAC_BYTEStoINT.3:= Byte0.3;
FUN_GTAC_BYTEStoINT.4:= Byte0.4;
FUN_GTAC_BYTEStoINT.5:= Byte0.5;
FUN_GTAC_BYTEStoINT.6:= Byte0.6;
FUN_GTAC_BYTEStoINT.7:= Byte0.7;

(*Byte 1 to Upper 8 bits of Int*)
FUN_GTAC_BYTEStoINT.8:= Byte1.0;
FUN_GTAC_BYTEStoINT.9:= Byte1.1;
FUN_GTAC_BYTEStoINT.10:= Byte1.2;
FUN_GTAC_BYTEStoINT.11:= Byte1.3;
FUN_GTAC_BYTEStoINT.12:= Byte1.4;
FUN_GTAC_BYTEStoINT.13:= Byte1.5;
FUN_GTAC_BYTEStoINT.14:= Byte1.6;
FUN_GTAC_BYTEStoINT.15:= Byte1.7;

END_FUNCTION

// ---- POUs/FBs/FB_SystemDiags20241206.TcPOU
(*FB for use gathering mother board data:
	Original Author(s): Chris Drees of Sodecia GTAC; 
------------------------------------------------------------------------------------------
REVISION NOTES:
	Version 20191210
	- Original Concept, c.drees
	Version 20241206
	- Corrected missing module read error, added in new module read fb type and did some general cleanup, b.lekx-toniolo
------------------------------------------------------------------------------------------
*)


FUNCTION_BLOCK FB_SystemDiags20241206
VAR_INPUT
    bRestart            :BOOL;               // flag to trigger restart of statemachine
END_VAR
VAR_OUTPUT
	HardwareDiag		:udt_HardwareDiags;
END_VAR
VAR
	sAmsNetId           :STRING := '';       //** ADS Net ID (local = '')    
    eState              :E_State;            // Enum with index for state machine     
    stMDP_Addr          : ST_MDP_Addr;        // structure will include all address parameters 
	
    uData               :UINT;               	// data storage for unsigned integer  
	iData				:INT;					//data storage for signed integer
	yData				:BYTE;					//Data Storage for Byte Data
	dData				:DINT;					//data Storage for Double Integer
	sData				:STRING;				//Data Storage for String Data   
 
    
    // FB instances
    fbReadMDPElement    : FB_MDP_ReadElement; // instance of FB for reading MDP element  
	fbIPCDiagReadParam	: FB_IPCDiag_ReadParameter;
	fbRegister     : FB_IPCDiag_Register;
	pBuffer			: DINT;

    // results of execution
    bError              : BOOL;               // error flag (indicator: error occured)
    nErrID              : UDINT;              // last error ID
	
	
	
END_VAR

(* 	
	The purpose of this function block is to replace the Motherboard Device that was present in TwinCAT2, due to changes between TC2 and TC3
	the motherboard device no longer exists and all data to be pulled for diagnostics must now use the MDP element.
	
	This Function Block is a large sequence of 25 steps, every two steps is one piece of data pulled from the MDP information.
*)


CASE eState OF
    0:               // initiate program parameters (if required)
        fbReadMDPElement(bExecute := FALSE);   	// ensure parameter 'bExecute' has FALSE state at startup 
		fbIPCDiagReadParam(bExecute := FALSE, fbRegister:= fbRegister);
		fbRegister(bExecute:= TRUE);				//Must be pre-called before referenced by fb_IPCDiag_ReadParameter Instance
        eState := 24;     							//Note, set this value to 26 for IPC that generate an error in steps 24 and 25 below

	// Attempt to Read CPU Temperature (uses newer FB from TC3_IPCDiag library) ------------------------------
	// Note, CPU Temp data is not be avail on all IPCs, if step 24 + 25 generates an error, set eState above to 26 to skip over and add "NA on this IPC" note to UI text field
    24:    
    	fbRegister(bExecute:= FALSE);								
	    IF NOT fbRegister.bBusy THEN     			// FB executed?
	        fbIPCDiagReadParam(
	            bExecute:= TRUE,               		
  	 			eParameterKey:= E_IPCDiag_ParameterKey.CPU_Temp,
    			sNetId:= '',
				fbRegister:= fbRegister
 				);                                
		END_IF;	
        eState := 25;  //** next state: process FB
		
	//Evaluate Response          
    25:                
        fbIPCDiagReadParam(bExecute := FALSE , fbRegister:= fbRegister);     
        IF NOT fbIPCDiagReadParam.bBusy THEN     // FB executed?
            IF fbIPCDiagReadparam.bError THEN    // Error?
                bError    := TRUE;             // set error flag
                nErrID    := fbIPCDiagReadParam.hrErrorCode; // store error id 
                eState    := 100; // finish state machine
            ELSE                               // set parameters for next steps
                bError    := FALSE;            // turn off error flag
				fbIPCDiagReadParam.GetParameter(ADR(pBuffer), SIZEOF(pBuffer)); //Call Method to retrieve data
                HardwareDiag.CpuTemp := DINT_TO_INT(pBuffer);            		//Store data to dedicated variable
                eState    := 26; //** next state 
            END_IF
        END_IF
	//---------------------------------------------------------		
	

	// Attempt to Read Fan Speed ------------------------------
    26:    
        stMDP_Addr.nArea    := INT_TO_BYTE(eMDP_Area_ConfigArea); //** set area address to "Config Area"
        stMDP_Addr.nTableId := 1;              //** table ID in module for "fan properties" table
        stMDP_Addr.nSubIdx  := 1;              //** subindex in table ID for "Fan RPM"                     
        
        fbReadMDPElement(
            bExecute    := TRUE,               // Flag: trigger execution of FB
            eModuleType := eMDP_ModT_Fan,      //** desired module type = CPU         
            stMDP_Addr  := stMDP_Addr,         // MDP address structure. Dynamic module ID added internally. 
            iModIdx     := 0,                  //** instance of desired module type (0 = first instance) 
            pDstBuf     := ADR(iData),         // buffer for storing data
            cbDstBufLen := SIZEOF(iData),      // length of buffer
            sAmsNetId   := sAmsNetId,          // AMS Net ID
            );                                 //** Note: fbReadMDPElement.tTimeOut must be > cycle time!

        eState := 27;  //** next state: process FB
 
	//Evaluate Response           
    27:                //** process FB: request CPU data
        fbReadMDPElement(bExecute := FALSE);   
        IF NOT fbReadMDPElement.bBusy THEN     // FB executed?
            IF fbReadMDPElement.bError THEN    // Error?
                bError    := TRUE;             // set error flag
                nErrID    := fbReadMDPElement.nErrID; // store error id (16#ECA60105 = BIOS or HW does 
                                               // not support this data (here: mainboard data))
                eState    := 100; // finish state machine
            ELSE                               // set parameters for next steps
                bError    := FALSE;            // turn off error flag
                HardwareDiag.FanSpeed := (iData);            //** store CPU usage in dedicated variable
                eState    := 28; //** next state 
            END_IF
        END_IF
	//-------------------------------------------------------------------	
		
	// Attempt to Mother Board Temperature ------------------------------
    28:    
        stMDP_Addr.nArea    := INT_TO_BYTE(eMDP_Area_ConfigArea); //** set area address to "Config Area"
        stMDP_Addr.nTableId := 1;              //** table ID in module for "mainboard information" table
        stMDP_Addr.nSubIdx  := 10;              //** subindex in table ID for "mainboard temperature (degC)"                     
        
        fbReadMDPElement(
            bExecute    := TRUE,               // Flag: trigger execution of FB
            eModuleType := eMDP_ModT_Mainboard,      //** desired module type = CPU         
            stMDP_Addr  := stMDP_Addr,         // MDP address structure. Dynamic module ID added internally. 
            iModIdx     := 0,                  //** instance of desired module type (0 = first instance) 
            pDstBuf     := ADR(iData),         // buffer for storing data
            cbDstBufLen := SIZEOF(iData),      // length of buffer
            sAmsNetId   := sAmsNetId,          // AMS Net ID
            );                                 //** Note: fbReadMDPElement.tTimeOut must be > cycle time!

        eState := 29;  //** next state: process FB
 
	//Evaluate Response           
    29:                //** process FB: request CPU data
        fbReadMDPElement(bExecute := FALSE);   
        IF NOT fbReadMDPElement.bBusy THEN     // FB executed?
            IF fbReadMDPElement.bError THEN    // Error?
                bError    := TRUE;             // set error flag
                nErrID    := fbReadMDPElement.nErrID; // store error id (16#ECA60105 = BIOS or HW does 
                                               // not support this data (here: mainboard data))
                eState    := 100; // finish state machine
            ELSE                               // set parameters for next steps
                bError    := FALSE;            // turn off error flag
                HardwareDiag.MboardTemp := (iData);            //Store data to dedicated variable
                eState    := 34; //** next state 
            END_IF
        END_IF
	//---------------------------------------------------------		
		
	// Attempt to Read 5 Volt supply actual voltage (in mV) ----------------------
    34:    
        stMDP_Addr.nArea    := INT_TO_BYTE(eMDP_Area_ConfigArea); //** set area address to "Config Area"
        stMDP_Addr.nTableId := 5;              //** table ID in module for "voltage information" table
        stMDP_Addr.nSubIdx  := 3;              //** subindex in table ID for "5v supply"                     
        
        fbReadMDPElement(
            bExecute    := TRUE,               // Flag: trigger execution of FB
            eModuleType := eMDP_ModT_Mainboard,      //** desired module type = CPU         
            stMDP_Addr  := stMDP_Addr,         // MDP address structure. Dynamic module ID added internally. 
            iModIdx     := 0,                  //** instance of desired module type (0 = first instance) 
            pDstBuf     := ADR(iData),         // buffer for storing data
            cbDstBufLen := SIZEOF(iData),      // length of buffer
            sAmsNetId   := sAmsNetId,          // AMS Net ID
            );                                 //** Note: fbReadMDPElement.tTimeOut must be > cycle time!

        eState := 35;  //** next state: process FB
            
	//Evaluate response
    35:                //** process FB: request CPU data
        fbReadMDPElement(bExecute := FALSE);    
        IF NOT fbReadMDPElement.bBusy THEN     // FB executed?
            IF fbReadMDPElement.bError THEN    // Error?
                bError    := TRUE;             // set error flag
                nErrID    := fbReadMDPElement.nErrID; // store error id (16#ECA60105 = BIOS or HW does 
                                               // not support this data (here: mainboard data))
                eState    := 100; // finish state machine
            ELSE                               // set parameters for next steps
                bError    := FALSE;            // turn off error flag
                HardwareDiag.Supply5V := (iData);            //Store data to dedicated variable
                eState    := 36; //** next state 
            END_IF
        END_IF
	//---------------------------------------------------------		
		
	// Attempt to Read 12 Volt supply actual voltage (in mV) ----------------------
    36:    
        stMDP_Addr.nArea    := INT_TO_BYTE(eMDP_Area_ConfigArea); //** set area address to "Config Area"
        stMDP_Addr.nTableId := 5;              //** table ID in module for "voltage information" table
        stMDP_Addr.nSubIdx  := 4;              //** subindex in table ID for "12v supply"                     
        
        fbReadMDPElement(
            bExecute    := TRUE,               // Flag: trigger execution of FB
            eModuleType := eMDP_ModT_Mainboard,      //** desired module type = CPU         
            stMDP_Addr  := stMDP_Addr,         // MDP address structure. Dynamic module ID added internally. 
            iModIdx     := 0,                  //** instance of desired module type (0 = first instance) 
            pDstBuf     := ADR(iData),         // buffer for storing data
            cbDstBufLen := SIZEOF(iData),      // length of buffer
            sAmsNetId   := sAmsNetId,          // AMS Net ID
            );                                 //** Note: fbReadMDPElement.tTimeOut must be > cycle time!

        eState := 37;  //** next state: process FB
            
	//Evaluate Response
    37:                //** process FB: request CPU data
        fbReadMDPElement(bExecute := FALSE);   
        IF NOT fbReadMDPElement.bBusy THEN     // FB executed?
            IF fbReadMDPElement.bError THEN    // Error?
                bError    := TRUE;             // set error flag
                nErrID    := fbReadMDPElement.nErrID; // store error id (16#ECA60105 = BIOS or HW does 
                                               // not support this data (here: mainboard data))
                eState    := 100; // finish state machine
            ELSE                               // set parameters for next steps
                bError    := FALSE;            // turn off error flag
                HardwareDiag.Supply12V := (iData);           //Store data to dedicated variable
                eState    := 40; //** next state 
            END_IF
        END_IF
	//---------------------------------------------------------		
		
	// Attempt to Read Battery Last Replace Date ----------------------
    40:    
        stMDP_Addr.nArea    := INT_TO_BYTE(eMDP_Area_ConfigArea); //** set area address to "Config Area"
        stMDP_Addr.nTableId := 1;              //** table ID in module for "UPS information" table
        stMDP_Addr.nSubIdx  := 17;              //** subindex in table ID for "battery replace date"                     
        
        fbReadMDPElement(
            bExecute    := TRUE,               // Flag: trigger execution of FB
            eModuleType := eMDP_ModT_UPS,      //** desired module type = CPU         
            stMDP_Addr  := stMDP_Addr,         // MDP address structure. Dynamic module ID added internally. 
            iModIdx     := 0,                  //** instance of desired module type (0 = first instance) 
            pDstBuf     := ADR(sData),         // buffer for storing data
            cbDstBufLen := SIZEOF(sData),      // length of buffer
            sAmsNetId   := sAmsNetId,          // AMS Net ID
            );                                 //** Note: fbReadMDPElement.tTimeOut must be > cycle time!

        eState := 41;  //** next state: process FB

	//Evaluate Response            
    41:                //** process FB: request CPU data
        fbReadMDPElement(bExecute := FALSE);   
        IF NOT fbReadMDPElement.bBusy THEN     // FB executed?
            IF fbReadMDPElement.bError THEN    // Error?
                bError    := TRUE;             // set error flag
                nErrID    := fbReadMDPElement.nErrID; // store error id (16#ECA60105 = BIOS or HW does 
                                               // not support this data (here: mainboard data))
                eState    := 100; // finish state machine
            ELSE                               // set parameters for next steps
                bError    := FALSE;            // turn off error flag
                HardwareDiag.BatteryReplaceDate := (sData);            //Store data to dedicated variable
                eState    := 42; //** next state 
            END_IF
        END_IF
	//---------------------------------------------------------		
		
	// Attempt to Read Battery Capacity ----------------------
    42:    
        stMDP_Addr.nArea    := INT_TO_BYTE(eMDP_Area_ConfigArea); //** set area address to "Config Area"
        stMDP_Addr.nTableId := 1;              //** table ID in module for "UPS Information" table
        stMDP_Addr.nSubIdx  := 10;              //** subindex in table ID for "battery capacity"                     
        
        fbReadMDPElement(
            bExecute    := TRUE,               // Flag: trigger execution of FB
            eModuleType := eMDP_ModT_UPS,      //** desired module type = CPU         
            stMDP_Addr  := stMDP_Addr,         // MDP address structure. Dynamic module ID added internally. 
            iModIdx     := 0,                  //** instance of desired module type (0 = first instance) 
            pDstBuf     := ADR(yData),         // buffer for storing data
            cbDstBufLen := SIZEOF(yData),      // length of buffer
            sAmsNetId   := sAmsNetId,          // AMS Net ID
            );                                 //** Note: fbReadMDPElement.tTimeOut must be > cycle time!

        eState := 43;  //** next state: process FB
		
 	//Evaluate Response           
    43:                //** process FB: request CPU data
        fbReadMDPElement(bExecute := FALSE);    
        IF NOT fbReadMDPElement.bBusy THEN     // FB executed?
            IF fbReadMDPElement.bError THEN    // Error?
                bError    := TRUE;             // set error flag
                nErrID    := fbReadMDPElement.nErrID; // store error id (16#ECA60105 = BIOS or HW does 
                                               // not support this data (here: mainboard data))
                eState    := 100; // finish state machine
            ELSE                               // set parameters for next steps
                bError    := FALSE;            // turn off error flag
                HardwareDiag.BatteryCapacity := (yData);            //Store data to dedicated variable
                eState    := 24; //** Done, restart 
            END_IF
        END_IF
	//---------------------------------------------------------		
		
	// Idle State in event of error (halt on error for easier capture) ----------------------
     100:                         // idle state 
         IF bRestart THEN                      // flag = TRUE -> restart state machine
            eState := 0;
   		 END_IF    
	//---------------------------------------------------------		
		
	// Default Case -----------------------------------------
	ELSE
    	eState := 100;                // capture undefined states 
	END_CASE 
	//--------------------------------------------------------

END_FUNCTION_BLOCK

// ---- POUs/FBs/FB_GTAC_ISxx_20241121.TcPOU
(*FB for use with Generic PDxx Panel conforming to SSCC V5xx

	Original Author(s):: Brent Lekx-Toniolo; 
------------------------------------------------------------------------------------------
REVISION NOTES:
	Version 20150812
		- Initial Concept, b.lekx-toniolo
	Version 20150928:
		- Added CoE reads fto gather EL6900 temperatue data, b.lekx-toniolo
	Version 20170303:
		- Split Power Relays to Estop and Safety Gate Relays, j.underhill
		- updated some unfinifshed sections of Eca cable breaks (more to come), j.underhill
	Version 20170307
		- Added Options to run split or non split relays and EP9224, b.lekx-toniolo
		- Added N999 (EP9224), b.lekx-toniolo
	Version 20170720
		- updated cable break for T05, j.vandongen
	Version 20180507
		- updated cable breaks, j.vandongen
	Version 20190924
		- changed T05 to EL6731, moved EK1110 to T06, j.vandongen (corrected comment 20221027, blt)
		- added Option input for EL6731, j.vandongen
	Version 20220907
		-Added N1000, N1001 to the discrete Image, C.drees
	Version 20241121
		-PD to IS rename, as per GH SSCC610 repo Issue#162, b.lekx-toniolo
		
------------------------------------------------------------------------------------------
*)

FUNCTION_BLOCK FB_GTAC_ISxx_20241121
	VAR_INPUT
		Enable_FB: BOOL;
		FB_In: udt_Generic_PD_20220906; (*Inputs to FB*)
	END_VAR

	VAR
(*Hardware Data Types*)
		(*Develop Discrete Nodes*)
		T01 AT %I*: udt_EK1100;						(*Ecat Bus Coupler*)
		T02_STAT AT %I*: udt_EL6900_STAT_20160426;	(*EL Safety CPU*)
		T02_CMD AT %Q*: udt_EL6900_CMD_20121204;
		T03 AT %I*: udt_EL1904_v2;						(*EL Safety Inputs*)
		T04 AT %I*: udt_EL2904RO_v2;					(*EL Safety Outputs, Set to "I" as this terminal is safety rated, therefore read only!*)
		T05 AT %I*: udt_EL6731;						(*EL Profibus Master*)
		T06 AT %I*: udt_EK1110_20150812;				(*Ecat Extension Terminal*)

		N01 AT %I*: udt_CU1128_20180507;				(*Ecat Junction Switch*)

		N999_STAT AT %I*: udt_EP9224_STAT_20161207;
		N999_CMD AT %Q*: udt_EP9224_CMD_20161207;
		N1000_STAT AT %I*: udt_EP9224_STAT_20161207;
		N1000_CMD AT %Q*: udt_EP9224_CMD_20161207;
		N1001_STAT AT %I*: udt_EP9224_STAT_20161207;
		N1001_CMD AT %Q*: udt_EP9224_CMD_20161207;		



(* Nodes States*)
		DiscreteNode_OK: BOOL;
		ProfiNode_OK: BOOL;

(*Cable Break Warning Flags*)
		ECatSlave_Cable_Breaks: UDINT;
		EK1100_NotPresent :BOOL;				(*Coupler is Not Present on Bus when expected*)
		EK1100_PortC_MissingLink: BOOL; 		(*Port C of EK1100 is OUT*)
		EK1110_PortB_MissingLink: BOOL; 		(*Port B of EK1110 is X1*)
		CU1128_PortD_MissingLink: BOOL;			(*SectionD Link 1 is for X2*)
		CU1128_PortD_MissingLink2: BOOL;		(*SectionD Link 2 is for X3*)
		CU1128_PortD_MissingLink3: BOOL;		(*SectionD Link 3 is for X6*)
		CU1128_PortB_MissingLink: BOOL;			(*SectionB Link 1 is for X4*)
		CU1128_PortB_MissingLink2: BOOL;		(*SectionB Link 2 is for X5*)
		CU1128_PortB_MissingLink3: BOOL;		(*SectionB Link 2 is for X7*)
		CU1128_PortC_MissingLink: BOOL;			(*SectionC is for Second section of Internal Fixtures X8*)
		N1000_Missing:BOOL; 					(*Second EP9224 Missing*)
		N1001_Missing:BOOL;						(*Third EP9224 Missing*)
			
(*CoE Read*)
		CoE_ReadFB_1: FB_EcCoESdoReadEx; 		(*FB to retrieve Data from terminals via CoE*)
		CoE_ReadBuffer_1: ARRAY [0..7] OF BYTE;	(*Variable, 8 bytes, for receiving data*)
		CoE_ReadErr_1: BOOL;					(*CoE Read Error Flag*)
		CoE_ReadErrID_1: UDINT;					(*CoE Read Error Identification*)
		EL6900_Overtemperature: BOOL;			(*Flag for result of CoE Read*)

(*Safety Internals*)
		Estop_Relays_On: BOOL;
		Estop_Relays_Off: BOOL;
		Gate_Relays_On: BOOL;
		Gate_Relays_Off: BOOL;
(*Standard Internals*)

		(*Fault Flags*)
		Estop_RelayFLT: BOOL;
		Gate_RelayFLT: BOOL;

	END_VAR

	VAR_OUTPUT
		FB_OK: BOOL;
		Discrete_Image: udt_ISxx_Image_20241121;
		Enable_SplitRelays AT%Q*: BOOL;				(*For mapping into Safety to Enable/Disable Second relay bank enable*)

	END_VAR



	(*Set FB_OK to True*)
	FB_OK:= TRUE;

(*$$$$$$$$$$$$$$$$$$$$$$$$$$$$$$$$$$$$$$$$$$$$$$$$Gather Status Of Hardware $$$$$$$$$$$$$$$$$$$$$$$$$$$$$$$$$$$$$$$$$$$$$$$$$$$$*)
	(*Discrete I/O Node*)
	IF (T01.InfoData.State=8) AND (T02_Stat.InfoData.State=8) AND (T03.InfoData.State=8) AND (T04.InfoData.State=8) AND ((T05.InfoData.State=8) OR NOT FB_In.Option_Enable_Pbus) AND (T06.InfoData.State=8)
		AND (N01.InfoData.State=8) AND (N01.InfoDataB.State=8) AND (N01.InfoDataC.State=8)
		AND ((N999_STAT.InfoData.State=8) OR FB_In.Option_EP9224_Count < 1)
		AND ((N1000_STAT.InfoData.State=8) OR FB_In.Option_EP9224_Count < 2)
		AND ((N1001_STAT.InfoData.State=8) OR FB_In.Option_EP9224_Count < 3)
		THEN DiscreteNode_OK:=TRUE;
	ELSE DiscreteNode_OK:=FALSE;
	END_IF;

	(*ProfiBus Node*)
	IF FB_In.Option_Enable_Pbus AND 
		(T05.InfoData.State<>0) AND		(*Ensure the termnal is at least alive*)
		(T05.Error=0) 
		THEN ProfiNode_OK:= TRUE;
	ELSE
		ProfiNode_OK:= FALSE;			
	END_IF;

	

	(*Develop Port Connection Warning Flags*)
	IF T01.InfoData.State=257  (*State Machine for Slave Not Present*)
		THEN EK1100_NotPresent:= TRUE;
	ELSE EK1100_NotPresent := FALSE;
	END_IF;

	IF T01.InfoData.State=17416 (*State Machine for Link Missing at Port C*)
		THEN EK1100_PortC_MissingLink:= TRUE; (*PortC is OUT Port*)
	ELSE EK1100_PortC_MissingLink := FALSE;
	END_IF;

	IF (T06.InfoData.State=9224)
		THEN EK1110_PortB_MissingLink:= TRUE;
	ELSE EK1110_PortB_MissingLink := FALSE;
	END_IF;


	IF ((N01.InfoData.State=33800) OR (N01.InfoData.State=41992))
		THEN CU1128_PortD_MissingLink:= TRUE;		(*PortD Attached at Port X2*)
	ELSE CU1128_PortD_MissingLink:= FALSE;
	END_IF;

	IF  ((N01.InfoData.State=9224) OR (N01.InfoData.State=41992))
		THEN CU1128_PortB_MissingLink:= TRUE;		(*PortB Attached at Port X3*)
	ELSE CU1128_PortB_MissingLink:= FALSE;
	END_IF;

	IF ((N01.InfoDataB.State=33800) OR (N01.InfoDataB.State=41992))
		THEN CU1128_PortD_MissingLink2:= TRUE;		(*PortD Attached at Port X4*)
	ELSE CU1128_PortD_MissingLink2:= FALSE;
	END_IF;

	IF  ((N01.InfoDataB.State=9224) OR (N01.InfoDataB.State=41992))
		THEN CU1128_PortB_MissingLink2:= TRUE;		(*PortB Attached at Port X5*)
	ELSE CU1128_PortB_MissingLink2:= FALSE;
	END_IF;

	IF ((N01.InfoDataC.State=33800) OR (N01.InfoDataC.State=41992)
		OR (N01.InfoDataC.State=50184) OR (N01.InfoDataC.State=58376))
		THEN CU1128_PortD_MissingLink3:= TRUE;		(*PortD Attached at Port X6*)
	ELSE CU1128_PortD_MissingLink3:= FALSE;
	END_IF;

	IF  ((N01.InfoDataC.State=9224) OR (N01.InfoDataC.State=25608)
		OR (N01.InfoDataC.State=41992) OR (N01.InfoDataC.State=58376))
		THEN CU1128_PortB_MissingLink3:= TRUE;		(*PortB Attached at Port X7*)
	ELSE CU1128_PortB_MissingLink3:= FALSE;
	END_IF;

	IF  ((N01.InfoDataC.State=17416) OR (N01.InfoDataC.State=25608)
		OR (N01.InfoDataC.State=50184) OR (N01.InfoDataC.State=58376))
		THEN CU1128_PortC_MissingLink:= TRUE;		(*PortC Attached at Port X8*)
	ELSE CU1128_PortC_MissingLink:= FALSE;
	END_IF;
	
	IF (N999_Stat.InfoData.State=9224) AND (FB_In.Option_EP9224_Count >1) (*State 9224 is missing link on port B*)
		THEN N1000_Missing:= TRUE;
	ELSE N1000_Missing := FALSE;
	END_IF;
	
	IF (N1000_Stat.InfoData.State=9224) AND (FB_In.Option_EP9224_Count >2) (*State 9224 is missing link on port B*)
		THEN N1001_Missing:= TRUE;
	ELSE N1001_Missing := FALSE;
	END_IF;

	(*Wrap up break Flags to Variable for shipment to UI*)
	ECatSlave_Cable_Breaks.0:= EK1100_NotPresent AND FB_In.Prev_EcatNode_Present;
	ECatSlave_Cable_Breaks.1:= EK1100_PortC_MissingLink;

	ECatSlave_Cable_Breaks.16:= EK1110_PortB_MissingLink; (*X1*)
	ECatSlave_Cable_Breaks.17:= CU1128_PortD_MissingLink; (*x2*)
	ECatSlave_Cable_Breaks.18:= CU1128_PortD_MissingLink2 (*x3*);
	ECatSlave_Cable_Breaks.19:= CU1128_PortD_MissingLink3; (*x4*)
	ECatSlave_Cable_Breaks.20:= CU1128_PortB_MissingLink; (*x5*)
	ECatSlave_Cable_Breaks.21:= CU1128_PortB_MissingLink2; (*x6*)
	ECatSlave_Cable_Breaks.22:= CU1128_PortB_MissingLink3; (*x7*)
	ECatSlave_Cable_Breaks.23:= CU1128_PortC_MissingLink; (*x8*)
	EcatSlave_Cable_Breaks.24:= N1000_Missing;
	EcatSlave_Cable_Breaks.25:= N1001_Missing;
	


	(*------------ CoE Reads ------------*)

	(*Read EL6900 Primaray Temperature Data*)

	(*FB Inputs*)
	CoE_ReadFB_1.bExecute:= FB_In.CoE_Read_Trigger
							AND (T02_Stat.InfoData.State=8);						(*Execute Upon Trigger*)
	CoE_ReadFB_1.sNetId:= FB_In.Ecat_Master_AmsNetID;
	CoE_ReadFB_1.nSlaveAddr:= T02_STAT.InfoData.AdsAddr.port;						(*Address of Ecat Slave being Read*)
	CoE_ReadFB_1.nIndex:= 16#FA80;												(*CANopen SDO Index of Object (FA80 = Hardware Diag Object)*)
	CoE_ReadFB_1.nSubIndex:= 16#01;												(*CANopen SDO SubIndex (Location from Index) of Object (1 = Primary Temperature)*)
	CoE_ReadFB_1.cbBufLen:= 8;													(*Limit on Receive Length (bytes)*)
	CoE_ReadFB_1.pDstBuf:= ADR(CoE_ReadBuffer_1);								(*Pointer to Receive Buffer*)
	CoE_ReadFB_1.tTimeout:= T#2s;												(*TImeout for Read*)
	CoE_ReadFB_1.bCompleteAccess:= TRUE;										(*Allow Complete Access to Full SDO Object*)

	(*Execute FB*)
	CoE_ReadFB_1();

	(*FB Outputs*)
	CoE_ReadErr_1:= CoE_ReadFB_1.bError;										(*Error Flag of Read*)
	CoE_ReadErrID_1:= CoE_ReadFB_1.nErrId;										(*Error ID of Read (See ADS Return Codes)*)

	(*Tranfer Data to Image*)
	IF (T02_Stat.InfoData.State=8) AND NOT CoE_ReadErr_1
		THEN
		T02_STAT.CoE_Temperature_1:= FUN_GTAC_BYTEStoINT(CoE_ReadBuffer_1[0],CoE_ReadBuffer_1[1]);	(*Grab bytes 0 and 1 of read buffer, this is Primary Temperature*)
		T02_STAT.CoE_Temperature_2:= FUN_GTAC_BYTEStoINT(CoE_ReadBuffer_1[2],CoE_ReadBuffer_1[3]);	(*Grab bytes 2 and 3 of read buffer, this is Secondary Temperature*)
	ELSE
		(*If Read Error, then blank data*)
		T02_STAT.CoE_Temperature_1:=0;
		T02_STAT.CoE_Temperature_2:=0;
	END_IF;

	(*Finally Evaluate Temperature Vs Upper Limit Restrictions*)
	IF (T02_STAT.CoE_Temperature_1>=90) OR (T02_STAT.CoE_Temperature_2>=90)
		THEN
		EL6900_Overtemperature:= TRUE;
	ELSE
		EL6900_Overtemperature:= FALSE;
	END_IF;


(*$$$$$$$$$$$$$$$$$$$$$$$$$$$$$$$$$$$$$$$$$$$$$ Gather Safety Inputs $$$$$$$$$$$$$$$$$$$$$$$$$$$$$$$$$$$$$$$$$$$$$$$$$$$$$$$$$*)

	(*Estop Relays (Contactors), Also Used as Power Relays in event of Option_Enable_SplitRelays being false*)
	Estop_Relays_On:= NOT T03.I.0;
	Estop_Relays_Off:= T03.I.0;

	(*Gate Relays (Contactors)*)
	IF FB_In.Option_Enable_SplitRelays
		THEN
		Gate_Relays_On:= NOT T03.I.1;
		Gate_Relays_Off:= T03.I.1;
	ELSE
		Gate_Relays_On:= FALSE;
		Gate_Relays_Off:= FALSE;
	END_IF;

(*$$$$$$$$$$$$$$$$$$$$$$$$$$$$$$$$$$$$$$$$$$$$$ Gather Standard Inputs $$$$$$$$$$$$$$$$$$$$$$$$$$$$$$$$$$$$$$$$$$$$$$$$$$$$$$$$$*)
	(*gather safety input data here*)
(*$$$$$$$$$$$$$$$$$$$$$$$$$$$$$$$$$$$$$$$$$$$$$ Internal Code $$$$$$$$$$$$$$$$$$$$$$$$$$$$$$$$$$$$$$$$$$$$$$$$$$$$$$$$$*)
	(*add internal code here*)
(*$$$$$$$$$$$$$$$$$$$$$$$$$$$$$$$$$$$$$$$$$$$$$$$$$$$ Faults $$$$$$$$$$$$$$$$$$$$$$$$$$$$$$$$$$$$$$$$$$$$$$$$$$$$$$$*)


	(*Estop/Power Relays EDM Fault*)
	Estop_RelayFLT:= ((T04.Q.0 AND NOT Estop_Relays_On) OR (NOT T04.Q.0 AND NOT Estop_Relays_Off)); (*Note, used as Power Relays if Split relay option is false*)

	(*Gate Relays EDM Fault*)
	IF FB_In.Option_Enable_SplitRelays
		THEN
		Gate_RelayFLT:= ((T04.Q.2 AND NOT Gate_Relays_On) OR (NOT T04.Q.2 AND NOT Gate_Relays_Off));
	ELSE
		Gate_RelayFLT:= FALSE;
	END_IF;

(*$$$$$$$$$$$$$$$$$$$$$$$$$$$$$$$$$$$$$$$$$$$$$$ Transfer Standard Outputs $$$$$$$$$$$$$$$$$$$$$$$$$$$$$$$$$$$$$$$$$$$*)
	(*Transfer I/O Images for Display On UI*)
	Discrete_Image.T01:=T01;
	Discrete_Image.T02_STAT:=T02_STAT;
	Discrete_Image.T03:=T03;
	Discrete_Image.T04:=T04;
	Discrete_Image.T05:=T05;
	Discrete_Image.T06:=T06;
	Discrete_Image.N01:=N01;

	Discrete_Image.N999_STAT:=N999_STAT;
	Discrete_Image.N999_CMD:=N999_CMD;
	Discrete_Image.N1000_STAT:=N1000_STAT;
	Discrete_Image.N1000_CMD:=N1000_CMD;
	Discrete_Image.N1001_STAT:=N1001_STAT;
	Discrete_Image.N1001_CMD:=N1001_CMD;
	
	(*Transfer Option Variables for Display on UI*)
	Discrete_Image.Option_Enable_SplitRelays:= FB_In.Option_Enable_SplitRelays;
	Discrete_Image.Option_EP9224_Count:= FB_In.Option_EP9224_Count;
	Discrete_Image.Option_Enable_Pbus:= FB_In.Option_Enable_Pbus;

	(*Transfer Split Relay Option to Physical Output*)
	Enable_SplitRelays:= FB_In.Option_Enable_SplitRelays;
	
(*$$$$$$$$$$$$$$$$$$$$$$$$$$$$$$$$$$$$$$$$$$$$$$ Transfer Safety Outputs $$$$$$$$$$$$$$$$$$$$$$$$$$$$$$$$$$$$$$$$$$$*)

(*Transfer Commands to Power Distribution Node Outputs*)
	(*Device Level*)
	N999_CMD.Device.Enable_Control_Via_Fieldbus:= FALSE;
	N999_CMD.Device.Global_Reset:= FB_In.Safety_RST;
	(*Channel1 Level*)
	N999_CMD.Channel1.Output_Us:= TRUE;
	N999_CMD.Channel1.Output_Up:= FB_In.Enable_Motion;
	N999_CMD.Channel1.Reset_Us:= FB_In.Safety_RST;
	N999_CMD.Channel1.Reset_Up:= FB_In.Safety_RST;
	(*Channel2Level*)
	N999_CMD.Channel2.Output_Us:= TRUE;
	N999_CMD.Channel2.Output_Up:= FB_In.Enable_Motion;
	N999_CMD.Channel2.Reset_Us:= FB_In.Safety_RST;
	N999_CMD.Channel2.Reset_Up:= FB_In.Safety_RST;
	(*Channel3Level*)
	N999_CMD.Channel3.Output_Us:= TRUE;
	N999_CMD.Channel3.Output_Up:= FB_In.Enable_Motion;
	N999_CMD.Channel3.Reset_Us:= FB_In.Safety_RST;
	N999_CMD.Channel3.Reset_Up:= FB_In.Safety_RST;
	(*Channel4Level*)
	N999_CMD.Channel4.Output_Us:= TRUE;
	N999_CMD.Channel4.Output_Up:= FB_In.Enable_Motion;
	N999_CMD.Channel4.Reset_Us:= FB_In.Safety_RST;
	N999_CMD.Channel4.Reset_Up:= FB_In.Safety_RST;

	(*Set All Safety Groups to Run*)
		T02_CMD.SGs_RUNSTOP:= TRUE;
	(*Reset Of Safety Group Errors*)
		T02_CMD.SGs_ERRAck:= FB_In.Safety_RST;
	(*Reset Only Used FBs With In Safety Group*)
		(*Reset of Estop, Safety Gate and Misc FBs*)
		T02_CMD.FBs_ControlPowerPB:= FB_In.Safety_RST;

END_FUNCTION_BLOCK

// ---- POUs/FBs/FB_GTAC_ICxx_20181023.TcPOU
(*FB for use with Generic ICxx Panel conforming to SSCC V5.xx

	Original Author(s): Brent Lekx-Toniolo/Rob Remillard of Sodecia GTAC.; 
------------------------------------------------------------------------------------------
REVISION NOTES:
	Version 1.0: August 2010
		- Initial Concept
	Version 20120607
		Changes from previous include:
			- Un-commented T14 Stat
	Version 20141202
			- Corrected Port B Cable Break Detect Flag, b.lekx-toniolo
	Version 20141205
			- Added SafetyGate_Latch_OK Variable, b.lekx-toniolo
	Version 20150120:
			- Added "previous ecat node ok" input for more accurate display of cable breaks, b.lekx-toniolo
	Version 20150326:
			- Added State checks for both X1 and X2 ports dissconnected on EK1122, b.lekx-toniolo
	Version 20150928:
			- Added CoE reads to gather EL6900 temperatue data, b.lekx-toniolo
			- Removed Main Relays as per new HW spec, b.lekx-toniolo
	Version 20170713
			- Added OP1_LC_Clear and OP2_LC_Clear bits for external control, j.vandongen
	Version 20171130
			- Added OP1_Yellow_Lamp_REQ and OP2_Yellow_Lamp_Req, j.vandongen
	Version 20181023
			- added provisions if a turntable is used, j.vandongen
------------------------------------------------------------------------------------------
*)

FUNCTION_BLOCK FB_GTAC_ICxx_20181023
	VAR_INPUT
		Enable_FB: BOOL;
		FB_In: udt_Generic_IC_20150928; (*Inputs to FB*)

		OP1_LC_Clear: BOOL;
		OP2_LC_Clear: BOOL;

		Turntable_Type: BOOL;

		Op1_At_Operator: BOOL;
		Op2_At_Operator: BOOL;

	END_VAR

	VAR
(*Hardware Data Types*)
		(*Develop Discrete Nodes*)
		T01 AT %I*: udt_EK1100;						(*Ecat Bus Coupler*)
		T02_STAT AT %I*: udt_EL6900_STAT_20160426;	(*EL Safety CPU*)
		T02_CMD AT %Q*: udt_EL6900_CMD_20121204;
		T03 AT %I*: udt_EL1904_v2;						(*EL Safety Inputs*)
		T04 AT %I*: udt_EL1904_v2;						(*EL Safety Inputs*)
		T05 AT %I*: udt_EL1904_v2;						(*EL Safety Inputs*)
		T06 AT %I*: udt_EL1904_v2;						(*EL Safety Inputs*)
		T07 AT %I*: udt_EL1904_v2;						(*EL Safety Inputs*)
		T08 AT %I*: udt_EL1904_v2;						(*EL Safety Inputs*)
		T09 AT %I*: udt_EL2904RO_v2;					(*EL Safety Outputs, Set to "I" as this terminal is safety rated, therefore read only!*)
		T10 AT %I*: udt_EL2904RO_v2;					(*EL Safety Outputs, Set to "I" as this terminal is safety rated, therefore read only!*)
		T11 AT %I*: udt_EL94xx;						(*EBUS Power Restoration*)
		T12 AT %I*: udt_EL1004_v2;						(*EL Inputs*)
		T13 AT %I*: udt_EL1004_v2;						(*EL Inputs*)
		T14 AT %Q*: udt_EL2008_v2;					(*EL Outputs, 8 Point*)
		T14_STAT AT %I*: udt_EL2008_STAT;			(*EL Output Card Status*)
		T15 AT %Q*: udt_EL2622;						(*EL Outputs, 2 Point*)
		T15_STAT AT %I*: udt_EL2622_STAT;			(*EL Output Card Status*)
		T16 AT%I*: udt_EK1122; 						(*ECAT Junction*)

(* Nodes States*)
		DiscreteNode_OK: BOOL;
		Ecat_Junction_OK: BOOL;
(*Cable Break Warning Flags*)
		ECatSlave_Cable_Breaks: UDINT;
		EK1100_NotPresent :BOOL;			(*Coupler is Not Present on Bus when expected*)
		EK1100_PortC_MissingLink: BOOL; 	(*Port C of EK1100 is OUT*)
		EK1122_PortD_MissingLink: BOOL; 	(*Port D of EK1122 is X1*)
		EK1122_PortB_MissingLink: BOOL;	(*Port B of EK1122 is X2*)
(*CoE Read*)
		CoE_ReadFB_1: FB_EcCoESdoReadEx; 		(*FB to retrieve Data from terminals via CoE*)
		CoE_ReadBuffer_1: ARRAY [0..7] OF BYTE;	(*Variable, 8 bytes, for receiving data*)
		CoE_ReadErr_1: BOOL;					(*CoE Read Error Flag*)
		CoE_ReadErrID_1: UDINT;					(*CoE Read Error Identification*)
		EL6900_Overtemperature: BOOL;			(*Flag for result of CoE Read*)

(*Safety Internals*)
		OP1_Estop_OK: BOOL;
		OP1_Cycle_Start: BOOL;
		OP1_HumanVertLC_Clear: BOOL;
		OP1_HumanHorizLC_Clear: BOOL;
		OP1_RobotVertLC_Clear: BOOL;
		OP1_Relays_On: BOOL;
		OP1_Relays_Off: BOOL;

		OP2_Estop_OK: BOOL;
		OP2_Cycle_Start: BOOL;
		OP2_HumanVertLC_Clear: BOOL;
		OP2_HumanHorizLC_Clear: BOOL;
		OP2_RobotVertLC_Clear: BOOL;
		OP2_Relays_On: BOOL;
		OP2_Relays_Off: BOOL;

		Main_Relays_On: BOOL;
		Main_Relays_Off: BOOL;

		SafetyGate_Latch_OK: BOOL;
(*Standard Internals*)
		Estop_PBs_OK: BOOL;
		OP1_AllHumanLCs_Clear: BOOL;
		OP2_AllHumanLCs_Clear: BOOL;
		Main_Air_Pressure_OK: BOOL;
		Loop_Indicies: ARRAY[0..9] OF INT:=[0]; (*Counters for For Loops*)
		OP1_Green_Lamp: BOOL;
		OP1_Yellow_Lamp: BOOL;
		OP1_Red_Lamp: BOOL;
		OP1_Audible: BOOL;
		OP2_Green_Lamp: BOOL;
		OP2_Yellow_Lamp: BOOL;
		OP2_Red_Lamp: BOOL;
		OP2_Audible: BOOL;

		Pulse_1S_FB: FB_Pulse_Generator;
		Pulse_1S: BOOL;
		Pulse_500ms_FB: FB_Pulse_Generator;
		Pulse_500ms: BOOL;
		Pulse_125ms_FB: FB_Pulse_Generator;
		Pulse_125ms: BOOL;

		KeyLOK_UnlockDelay_TMR: TON;

		(*Fault Flags*)
		OP1_RelayFLT: BOOL;
		OP2_RelayFLT: BOOL;
		Main_RelayFLT: BOOL;

END_VAR

	VAR_OUTPUT
		FB_OK: BOOL;
		Discrete_Image: udt_ICxx_Image;
		OP1_Enable_Motion: BOOL;
		OP2_Enable_Motion: BOOL;

	END_VAR

	(*Set FB_OK to True*)
	FB_OK:= TRUE;
(*$$$$$$$$$$$$$$$$$$$$$$$$$$$$$$$$$$$$$$$$$$$$$$$$Gather Status Of Hardware $$$$$$$$$$$$$$$$$$$$$$$$$$$$$$$$$$$$$$$$$$$$$$$$$$$$*)
	(*Discrete I/O Node*)
	IF T01.InfoData.State=8 AND T02_Stat.InfoData.State=8 AND T03.InfoData.State=8 AND T04.InfoData.State=8 AND T05.InfoData.State=8
		AND T06.InfoData.State=8 AND T07.InfoData.State=8 AND T08.InfoData.State=8 AND T09.InfoData.State=8 AND T10.InfoData.State=8
		AND T11.InfoData.State=8 AND T12.InfoData.State=8 AND T13.InfoData.State=8 AND T14_Stat.InfoData.State=8 AND T15_Stat.InfoData.State=8
		AND T16.InfoData.State=8

		THEN DiscreteNode_OK:=TRUE;
	ELSE DiscreteNode_OK:=FALSE;
	END_IF;
	(*EtherCAT 2 Port Junction, For Interface to OP Fixtures*)
	IF T16.InfoData.State=8
		THEN Ecat_Junction_OK:=TRUE;
	ELSE Ecat_Junction_OK:=FALSE;
	END_IF;

	(*Develop Port Connection Warning Flags*)
	IF T01.InfoData.State=257  (*State Machine for Slave Not Present*)
		THEN EK1100_NotPresent:= TRUE;
	ELSE EK1100_NotPresent := FALSE;
	END_IF;

	IF T01.InfoData.State=17416 (*State Machine for Link Missing at Port C*)
		THEN EK1100_PortC_MissingLink:= TRUE; (*PortC is OUT Port*)
	ELSE EK1100_PortC_MissingLink := FALSE;
	END_IF;


	IF (T16.InfoData.State=-31736) (*State Machine for Link Missing at Port D (0xA8408)*)
		OR (T16.InfoData.State=-23544) (*State Machine for Link Missing at Port D and Port B (0xA408)*)
		THEN EK1122_PortD_MissingLink:= TRUE; (*Port D is X1 Port*)
	ELSE EK1122_PortD_MissingLink := FALSE;
	END_IF;

	IF (T16.InfoData.State=9224) (*State Machine for Link Missing at Port B (0x2408)*)
		OR (T16.InfoData.State=-23544) (*State Machine for Link Missing at Port D and Port B (0xA408)*)
		THEN EK1122_PortB_MissingLink:= TRUE; (*Port B is X2 Port*)
	ELSE EK1122_PortB_MissingLink := FALSE;
	END_IF;

	(*Wrap up break Flags to Variable for shipment to UI*)
	ECatSlave_Cable_Breaks.0:= EK1100_NotPresent AND FB_In.Prev_EcatNode_Present;
	ECatSlave_Cable_Breaks.1:= EK1100_PortC_MissingLink;
	ECatSlave_Cable_Breaks.16:=EK1122_PortD_MissingLink;
	ECatSlave_Cable_Breaks.17:=EK1122_PortB_MissingLink;

	(*------------ CoE Reads ------------*)

	(*Read EL6900 Primaray Temperature Data*)

	(*FB Inputs*)
	CoE_ReadFB_1.bExecute:= FB_In.CoE_Read_Trigger
							AND (T02_Stat.InfoData.State=8);						(*Execute Upon Trigger*)
	CoE_ReadFB_1.sNetId:= FB_In.Ecat_Master_AmsNetID;
	CoE_ReadFB_1.nSlaveAddr:= T02_STAT.InfoData.AdsAddr.port;						(*Address of Ecat Slave being Read*)
	CoE_ReadFB_1.nIndex:= 16#FA80;												(*CANopen SDO Index of Object (FA80 = Hardware Diag Object)*)
	CoE_ReadFB_1.nSubIndex:= 16#01;												(*CANopen SDO SubIndex (Location from Index) of Object (1 = Primary Temperature)*)
	CoE_ReadFB_1.cbBufLen:= 8;													(*Limit on Receive Length (bytes)*)
	CoE_ReadFB_1.pDstBuf:= ADR(CoE_ReadBuffer_1);								(*Pointer to Receive Buffer*)
	CoE_ReadFB_1.tTimeout:= T#2s;												(*TImeout for Read*)
	CoE_ReadFB_1.bCompleteAccess:= TRUE;										(*Allow Complete Access to Full SDO Object*)

	(*Execute FB*)
	CoE_ReadFB_1();

	(*FB Outputs*)
	CoE_ReadErr_1:= CoE_ReadFB_1.bError;										(*Error Flag of Read*)
	CoE_ReadErrID_1:= CoE_ReadFB_1.nErrId;										(*Error ID of Read (See ADS Return Codes)*)

	(*Tranfer Data to Image*)
	IF (T02_Stat.InfoData.State=8) AND NOT CoE_ReadErr_1
		THEN
		T02_STAT.CoE_Temperature_1:= FUN_GTAC_BYTEStoINT(CoE_ReadBuffer_1[0],CoE_ReadBuffer_1[1]);	(*Grab bytes 0 and 1 of read buffer, this is Primary Temperature*)
		T02_STAT.CoE_Temperature_2:= FUN_GTAC_BYTEStoINT(CoE_ReadBuffer_1[2],CoE_ReadBuffer_1[3]);	(*Grab bytes 2 and 3 of read buffer, this is Secondary Temperature*)
	ELSE
		(*If Read Error, then blank data*)
		T02_STAT.CoE_Temperature_1:=0;
		T02_STAT.CoE_Temperature_2:=0;
	END_IF;

	(*Finally Evaluate Temperature Vs Upper Limit Restrictions*)
	IF (T02_STAT.CoE_Temperature_1>=90) OR (T02_STAT.CoE_Temperature_2>=90)
		THEN
		EL6900_Overtemperature:= TRUE;
	ELSE
		EL6900_Overtemperature:= FALSE;
	END_IF;


(*$$$$$$$$$$$$$$$$$$$$$$$$$$$$$$$$$$$$$$$$$$$$ Gather Standard Inputs $$$$$$$$$$$$$$$$$$$$$$$$$$$$$$$$$$$$$$$$$$$$$$$$$$$$$$$$*)

	(*Air Pressure Switch*)
	Main_Air_Pressure_OK:= T12.I.0;

(*$$$$$$$$$$$$$$$$$$$$$$$$$$$$$$$$$$$$$$$$$$$$$ Gather Safety Inputs $$$$$$$$$$$$$$$$$$$$$$$$$$$$$$$$$$$$$$$$$$$$$$$$$$$$$$$$$*)
	(*OP1 Safety Status*)
	OP1_Estop_OK:= T03.I.0 AND T03.I.1;
	OP1_Cycle_Start:= T03.I.3;
	OP1_HumanVertLC_Clear:= T04.I.0 AND T04.I.1;
	OP1_HumanHorizLC_Clear:= T04.I.2 AND T04.I.3;
	OP1_RobotVertLC_Clear:= T05.I.0 AND T05.I.1;
	OP1_Relays_On:= NOT T05.I.3 AND T09.Q.0 AND T09.Q.1;
	OP1_Relays_Off:= T05.I.3;

	(*OP2 Safety Status*)
	OP2_Estop_OK:= T06.I.0 AND T06.I.1;
	OP2_Cycle_Start:= T06.I.3;
	OP2_HumanVertLC_Clear:= T07.I.0 AND T07.I.1;
	OP2_HumanHorizLC_Clear:= T07.I.2 AND T07.I.3;
	OP2_RobotVertLC_Clear:= T08.I.0 AND T08.I.1;
	OP2_Relays_On:= NOT T08.I.3 AND T10.Q.0 AND T10.Q.1;
	OP2_Relays_Off:= T08.I.3;

	(*Main Relay Status*)
	Main_Relays_On:= FALSE;
	Main_Relays_Off:= FALSE;

	(*Estop Status Of Area*)
	Estop_PBs_Ok:= OP1_Estop_OK AND OP2_Estop_Ok;

	(*SafetyGate Latch Status*)
	SafetyGate_Latch_Ok:= T03.I.2 AND T08.I.2;

(*$$$$$$$$$$$$$$$$$$$$$$$$$$$$$$$$$$$$$$$$$$$$$ Internal Code $$$$$$$$$$$$$$$$$$$$$$$$$$$$$$$$$$$$$$$$$$$$$$$$$$$$$$$$$*)
	(*Pulse Generators*)
		(*1 Second On and Off Time*)
		Pulse_1S_FB.On_Time:=T#1.0S;
		Pulse_1S_FB.Off_Time:=T#1.0S;
		Pulse_1S_FB();
		Pulse_1S:=Pulse_1S_FB.Wave;
		(*0.5 Second On and Off Time*)
		Pulse_500ms_FB.On_Time:=T#500ms;
		Pulse_500ms_FB.Off_Time:=T#500ms;
		Pulse_500ms_FB();
		Pulse_500ms:=Pulse_500ms_FB.Wave;
		(*0.25 Second On and Off Time*)
		Pulse_125ms_FB.On_Time:=T#125ms;
		Pulse_125ms_FB.Off_Time:=T#125ms;
		Pulse_125ms_FB();
		Pulse_125ms:=Pulse_125ms_FB.Wave;

	(*Gather Light Curtain Status*)
	OP1_AllHumanLCs_Clear:= OP1_LC_Clear;
	OP2_AllHumanLCs_Clear:= OP2_LC_Clear;

	(*Control Of Operator Station Lamps*)
	(*OP1*)
		(*Green Lamp*)
		OP1_Green_Lamp:=  FB_In.Estops_OK AND FB_In.Safety_Gates_Ok
					AND ((NOT Turntable_Type AND FB_In.OP1_Green_LampReq AND NOT FB_In.OP1_Red_LampReq)
					OR (Turntable_Type  AND Op1_At_Operator AND FB_In.OP1_Green_LampReq AND NOT FB_In.OP1_Red_LampReq)
					OR (Turntable_Type  AND Op2_At_Operator AND FB_In.OP2_Green_LampReq AND NOT FB_In.OP2_Red_LampReq));

		(*Yellow Lamp*)
		IF  FB_In.Estops_OK AND FB_in.Safety_Gates_Ok
			AND (( NOT Turntable_Type AND OP1_AllHumanLCs_Clear AND NOT OP1_Relays_On AND FB_In.OP1_Yellow_LampReq)
			OR (Turntable_Type AND Op1_At_Operator AND OP1_AllHumanLCs_Clear AND NOT OP1_Relays_On AND FB_In.OP1_Yellow_LampReq)
			OR (Turntable_Type AND Op2_At_Operator AND OP2_AllHumanLCs_Clear AND NOT OP2_Relays_On AND FB_In.OP2_Yellow_LampReq))
			THEN
				OP1_Yellow_Lamp:= Pulse_500ms;
		ELSIF NOT OP1_AllHumanLCs_Clear AND FB_In.Estops_OK
			THEN
				OP1_Yellow_Lamp:= TRUE;
		ELSE
				OP1_Yellow_Lamp:= FALSE;
		END_IF;

		(*Red Lamp*)
		IF NOT FB_IN.Estops_OK
			AND ((NOT Turntable_Type AND Op1_Estop_OK)
			OR (Turntable_Type  AND Op1_At_Operator AND OP1_Estop_Ok)
			OR (Turntable_Type  AND Op2_At_Operator AND OP2_Estop_Ok))
			THEN
				OP1_Red_Lamp:= TRUE;
		ELSIF NOT FB_IN.Estops_OK
			AND ((NOT Turntable_Type AND NOT Op1_Estop_OK)
			OR (Turntable_Type  AND Op1_At_Operator AND NOT OP1_Estop_Ok)
			OR (Turntable_Type  AND Op2_At_Operator AND NOT OP2_Estop_Ok))
			THEN
				OP1_Red_Lamp:= Pulse_500ms;
		ELSIF NOT FB_In.Safety_Gates_Ok AND FB_In.Estops_OK
			THEN
				OP1_Red_Lamp:= Pulse_500ms;
		ELSIF FB_In.Estops_OK
			AND ((NOT Turntable_Type AND FB_In.OP1_Red_LampReq)
			OR (Turntable_Type  AND Op1_At_Operator AND  FB_In.OP1_Red_LampReq)
			OR (Turntable_Type  AND Op2_At_Operator AND  FB_In.OP2_Red_LampReq))
			THEN
				OP1_Red_Lamp:= Pulse_125ms;
		ELSE
				OP1_Red_Lamp:= FALSE;
		END_IF;

		(*Audible*)
		OP1_Audible:= ((NOT Turntable_Type AND FB_In.OP1_Audible_Req)
				OR (Turntable_Type  AND Op1_At_Operator AND FB_In.OP1_Audible_Req)
				OR (Turntable_Type  AND Op2_At_Operator AND FB_In.OP2_Audible_Req));


	(*OP2*)
		(*Green Lamp*)
		OP2_Green_Lamp:=  FB_In.Estops_OK AND FB_In.Safety_Gates_Ok
					AND ((NOT Turntable_Type AND FB_In.OP2_Green_LampReq AND NOT FB_In.OP2_Red_LampReq)
					OR (Turntable_Type  AND Op1_At_Operator AND FB_In.OP1_Green_LampReq AND NOT FB_In.OP1_Red_LampReq)
					OR (Turntable_Type  AND Op2_At_Operator AND FB_In.OP2_Green_LampReq AND NOT FB_In.OP2_Red_LampReq));

		(*Yellow Lamp*)
		IF  FB_In.Estops_OK AND FB_in.Safety_Gates_Ok
			AND (( NOT Turntable_Type AND OP2_AllHumanLCs_Clear AND NOT OP2_Relays_On AND FB_In.OP2_Yellow_LampReq)
			OR (Turntable_Type AND Op1_At_Operator AND OP1_AllHumanLCs_Clear AND NOT OP1_Relays_On AND FB_In.OP1_Yellow_LampReq)
			OR (Turntable_Type AND Op2_At_Operator AND OP2_AllHumanLCs_Clear AND NOT OP2_Relays_On AND FB_In.OP2_Yellow_LampReq))
			THEN
				OP2_Yellow_Lamp:= Pulse_500ms;
		ELSIF NOT OP2_AllHumanLCs_Clear AND FB_In.Estops_OK
			THEN
				OP2_Yellow_Lamp:= TRUE;
		ELSE
				OP2_Yellow_Lamp:= FALSE;
		END_IF;

		(*Red Lamp*)
		IF NOT FB_IN.Estops_OK
			AND ((NOT Turntable_Type AND Op2_Estop_OK)
			OR (Turntable_Type  AND Op1_At_Operator AND OP1_Estop_Ok)
			OR (Turntable_Type  AND Op2_At_Operator AND OP2_Estop_Ok))
			THEN
				OP2_Red_Lamp:= TRUE;
		ELSIF NOT FB_IN.Estops_OK
			AND ((NOT Turntable_Type AND NOT Op2_Estop_OK)
			OR (Turntable_Type  AND Op1_At_Operator AND NOT OP1_Estop_Ok)
			OR (Turntable_Type  AND Op2_At_Operator AND NOT OP2_Estop_Ok))
			THEN
				OP2_Red_Lamp:= Pulse_500ms;
		ELSIF NOT FB_In.Safety_Gates_Ok AND FB_In.Estops_OK
			THEN
				OP2_Red_Lamp:= Pulse_500ms;
		ELSIF FB_In.Estops_OK
			AND ((NOT Turntable_Type AND FB_In.OP2_Red_LampReq)
			OR (Turntable_Type  AND Op1_At_Operator AND  FB_In.OP1_Red_LampReq)
			OR (Turntable_Type  AND Op2_At_Operator AND  FB_In.OP2_Red_LampReq))
			THEN
				OP2_Red_Lamp:= Pulse_125ms;
		ELSE
				OP2_Red_Lamp:= FALSE;
		END_IF;

		(*Audible*)
		OP2_Audible:= ((NOT Turntable_Type AND FB_In.OP2_Audible_Req)
				OR (Turntable_Type  AND Op1_At_Operator AND FB_In.OP1_Audible_Req)
				OR (Turntable_Type  AND Op2_At_Operator AND FB_In.OP2_Audible_Req));



	(*Handle LOK Release Requests*)
	KeyLOK_UnlockDelay_TMR.PT:= T#1.5s;
	KeyLOK_UnlockDelay_TMR();
	IF FB_In.Output_Req1
		THEN
		KeyLOK_UnlockDelay_TMR.IN:=TRUE;
	ELSE
		KeyLOK_UnlockDelay_TMR.IN:=FALSE;
	END_IF;




(*$$$$$$$$$$$$$$$$$$$$$$$$$$$$$$$$$$$$$$$$$$$$$$$$$$$ Faults $$$$$$$$$$$$$$$$$$$$$$$$$$$$$$$$$$$$$$$$$$$$$$$$$$$$$$$*)

OP1_RelayFLT:= ((T09.Q.0 AND NOT OP1_Relays_On) OR (NOT T09.Q.0 AND NOT OP1_Relays_Off));
OP2_RelayFLT:= ((T10.Q.0 AND NOT OP2_Relays_On) OR (NOT T10.Q.0 AND NOT OP2_Relays_Off));
Main_RelayFLT:= FALSE;

(*$$$$$$$$$$$$$$$$$$$$$$$$$$$$$$$$$$$$$$$$$$$$$$ Transfer Standard Outputs $$$$$$$$$$$$$$$$$$$$$$$$$$$$$$$$$$$$$$$$$$$*)
	(*Transfer I/O Images for Display On HMI*)
	Discrete_Image.T01:=T01;
	Discrete_Image.T02_STAT:=T02_STAT;
	Discrete_Image.T03:=T03;
	Discrete_Image.T04:=T04;
	Discrete_Image.T05:=T05;
	Discrete_Image.T06:=T06;
	Discrete_Image.T07:=T07;
	Discrete_Image.T08:=T08;
	Discrete_Image.T09:=T09;
	Discrete_Image.T10:=T10;
	Discrete_Image.T11:=T11;
	Discrete_Image.T12:=T12;
	Discrete_Image.T13:=T13;
	Discrete_Image.T14:=T14;
	Discrete_Image.T14_STAT:= T14_STAT;
	Discrete_Image.T15:=T15;
	Discrete_Image.T15_STAT:= T15_STAT;
	Discrete_Image.T16:=T16;

(*Transfer Commands to Discrete Node Outputs*)
	T14.Q.0:= OP1_Green_Lamp;			(*OP1 Green Lamp*)
	T14.Q.1:= OP1_Yellow_Lamp;			(*OP1 Yellow Lamp*)
	T14.Q.2:= OP1_Red_Lamp;				(*OP1 Red Lamp*)
	T14.Q.3:= OP1_Audible;				(*OP1 Audible "Buzzer"*)
	T14.Q.4:= OP2_Green_Lamp;			(*OP2 Green Lamp*)
	T14.Q.5:= OP2_Yellow_Lamp;			(*OP2 Yellow Lamp*)
	T14.Q.6:= OP2_Red_Lamp;				(*OP2 Red Lamp*)
	T14.Q.7:= OP2_Audible;				(*OP2 Audible "Buzzer"*)

	T15.Q0:= KeyLOK_UnlockDelay_TMR.Q;	(*EL2622 Output1*)
	T15.Q1:= FB_In.Output_Req2;			(*EL2622 Output2*)


(*$$$$$$$$$$$$$$$$$$$$$$$$$$$$$$$$$$$$$$$$$$$$$$ Transfer Safety Outputs $$$$$$$$$$$$$$$$$$$$$$$$$$$$$$$$$$$$$$$$$$$*)
	(*Transfer Enable_Motions for use by sub Components*)
		OP1_Enable_Motion:= (NOT Turntable_Type AND OP1_Relays_On AND OP1_AllHumanLCs_Clear)
				OR (Turntable_Type  AND Op1_At_Operator AND OP1_Relays_On AND OP1_AllHumanLCs_Clear)
				OR (Turntable_Type  AND Op2_At_Operator AND OP1_Relays_On);
		OP2_Enable_Motion:= (NOT Turntable_Type AND OP2_Relays_On AND OP2_AllHumanLCs_Clear)
				OR (Turntable_Type  AND Op1_At_Operator AND OP2_Relays_On)
				OR (Turntable_Type  AND Op2_At_Operator AND OP2_Relays_On AND OP2_AllHumanLCs_Clear);

	(*Set All Safety Groups to Run*)
		T02_CMD.SGs_RUNSTOP:= TRUE;
	(*Reset Of Safety Group Errors*)
		T02_CMD.SGs_ERRAck:= FB_In.Safety_RST;
	(*Reset Only Used FBs With In Safety Group*)
		(*Reset of Estop, Safety Gate and Misc FBs*)
		T02_CMD.FBs_ControlPowerPB:= FB_In.Safety_RST;

END_FUNCTION_BLOCK

// ---- POUs/FBs/FB_Pulse_Generator.TcPOU

(*Generic Pulse Generator to Create Adjustable Pulse WaveForm*)
FUNCTION_BLOCK FB_Pulse_Generator
VAR_INPUT
	On_Time: TIME;
	Off_Time: TIME;
END_VAR

VAR
	Internal_On_TMR: TON;
	Internal_Duty_Cycle: BYTE;
	Internal_Off_TMR: TON;
	Internal_Wave: BOOL;
END_VAR

VAR_OUTPUT
	Wave: BOOL;
END_VAR

(*Estabish Timer Data*)

	Internal_On_TMR.PT:=On_Time;
	Internal_Off_TMR.PT:=Off_Time;
	Internal_On_TMR();
	Internal_Off_TMR();

(*Generate Pulse*)
	(*Pulse High*)
	IF NOT Internal_Off_TMR.IN
		THEN
			Internal_On_TMR.IN:=TRUE;
			Internal_Wave:=TRUE;
	END_IF;
	IF Internal_On_TMR.Q
		THEN
			Internal_On_TMR.IN:=FALSE;
			Internal_Off_TMR.IN:= TRUE;
	END_IF;

	(*Pulse Low*)
	IF NOT Internal_On_TMR.IN
		THEN
			Internal_Wave:=FALSE;
	END_IF;

	IF Internal_Off_TMR.Q
		THEN
			Internal_Off_TMR.IN:=FALSE;
	END_IF;

(*Transfer Output*)
	Wave:=Internal_Wave;

END_FUNCTION_BLOCK

